// TIA Portal V20 program export: 22 tag tables, 10 data types, 20 data blocks, 41 code blocks (in call order from the OBs), 25 instance data blocks

VAR_GLOBAL   // PLC tag table "Cabinet13"
   Sz13_Column_Red AT %Q1201.2 : Bool;
   Sz13_Column_Buzzer AT %Q1201.4 : Bool;
   Sz13_Column_Green AT %Q1200.6 : Bool;
   Sz13_Column_Yellow AT %Q1201.0 : Bool;
END_VAR

VAR_GLOBAL   // PLC tag table "Cabinet14"
   Sz14_Column_Buzzer AT %Q1201.5 : Bool;
   Sz14_Column_Red AT %Q1201.3 : Bool;
   Sz14_Column_Yellow AT %Q1201.1 : Bool;
   Sz14_Column_Green AT %Q1200.7 : Bool;
END_VAR

VAR_GLOBAL   // PLC tag table "Cabinet_1"
   Sz1_St25_SenA AT %I1100.0 : Bool;
   Sz1_St25_SenB AT %I1100.1 : Bool;
   Sz1_St25_SenC AT %I1100.2 : Bool;
   Sz1_St25_SenD AT %I1100.3 : Bool;
   Sz1_St26_SenA AT %I1100.4 : Bool;
   Sz1_St26_SenB AT %I1100.5 : Bool;
   Sz1_St26_SenC AT %I1100.6 : Bool;
   Sz1_St26_SenD AT %I1100.7 : Bool;
   Sz1_St23_SenA AT %I1101.0 : Bool;
   Sz1_St23_SenB AT %I1101.1 : Bool;
   Sz1_St23_SenC AT %I1101.2 : Bool;
   Sz1_St23_SenD AT %I1101.3 : Bool;
   Sz1_St24_SenA AT %I1101.4 : Bool;
   Sz1_St24_SenB AT %I1101.5 : Bool;
   Sz1_St24_SenC AT %I1101.6 : Bool;
   Sz1_St24_SenD AT %I1101.7 : Bool;
   Sz1_Button_ST25_ST26 AT %I1102.0 : Bool;
   Sz1_Button_ST26_ST27 AT %I1102.1 : Bool;
   Sz1_Button_ST24_ST23 AT %I1102.2 : Bool;
   Sz1_Button_ST23_ST22 AT %I1102.3 : Bool;
   Sz1_Button_ST24_Seq_Backward AT %I1102.4 : Bool;
   Sz1_Button_ST24_Seq_Forward AT %I1102.5 : Bool;
   Sz1_Button_ST25_Seq_Backward AT %I1102.6 : Bool;
   Sz1_Button_ST25_Seq_Forward AT %I1102.7 : Bool;
   Sz1_Button_ST23_Seq_Forward AT %I1103.0 : Bool;
   Sz1_Button_SS_Down AT %I1103.1 : Bool;
   Sz1_Button_SS_Up AT %I1103.2 : Bool;
   Sz1_Button_SS_Drive_ST25 AT %I1103.3 : Bool;
   Sz1_Button_SS_Drive_ST24 AT %I1103.4 : Bool;
   Sz1_Button_SS_Drive_ST17 AT %I1103.5 : Bool;
   Sz1_Button_SS_Drive_ST14 AT %I1103.6 : Bool;
   "Reserved(1)" AT %I1103.7 : Bool;
   Sz1_Safety1_1 AT %I1150.0 : Bool;
   Sz13_Safety1_1 AT %I1150.1 : Bool;
   "Reserved(12)" AT %I1150.2 : Bool;
   "Reserved(13)" AT %I1150.3 : Bool;
   Sz1_Safety1_2 AT %I1150.4 : Bool;
   Sz13_Safety1_2 AT %I1150.5 : Bool;
   "Reserved(15)" AT %I1150.6 : Bool;
   "Reserved(16)" AT %I1150.7 : Bool;
   "Reserved(17)" AT %I1151.0 : Bool;
   "Reserved(18)" AT %I1151.1 : Bool;
   "Reserved(19)" AT %I1151.2 : Bool;
   "Reserved(20)" AT %I1151.3 : Bool;
   "Reserved(21)" AT %I1151.4 : Bool;
   "Reserved(22)" AT %I1151.5 : Bool;
   "Reserved(23)" AT %I1151.6 : Bool;
   "Reserved(24)" AT %I1151.7 : Bool;
   Sz1_Button_LED_ST25_ST26 AT %Q1100.0 : Bool;
   Sz1_Button_LED_ST26_ST27 AT %Q1100.1 : Bool;
   Sz1_Button_LED_ST24_ST23 AT %Q1100.2 : Bool;
   Sz1_Button_LED_ST23_ST22 AT %Q1100.3 : Bool;
   Sz1_Button_LED_Hyd_Up AT %Q1100.4 : Bool;
   Sz1_Button_LED_Hyd_Down AT %Q1100.5 : Bool;
   Sz1_Button_LED_Air_Up AT %Q1100.6 : Bool;
   Sz1_Button_LED_Air_Down AT %Q1100.7 : Bool;
   Sz1_Button_LED_Wibration AT %Q1101.0 : Bool;
   Sz1_Button_LED_SS_Down AT %Q1101.1 : Bool;
   Sz1_Button_LED_SS_Up AT %Q1101.2 : Bool;
   Sz1_Button_LED_SS_Drive_ST25 AT %Q1101.3 : Bool;
   Sz1_Button_LED_SS_Drive_ST24 AT %Q1101.4 : Bool;
   Sz1_Button_LED_SS_Drive_ST17 AT %Q1101.5 : Bool;
   Sz1_Button_LED_SS_Drive_ST14 AT %Q1101.6 : Bool;
   Reserved AT %Q1101.7 : Bool;
   Sz1_Button_LED_Centering_ST23 AT %Q1102.0 : Bool;
   Sz1_Button_LED_Centering_ST22 AT %Q1102.1 : Bool;
   "Reserved(5)" AT %Q1102.2 : Bool;
   "Reserved(6)" AT %Q1102.3 : Bool;
   Sz1_Button_LED_ST23_Seq_Backward AT %Q1102.4 : Bool;
   ST23_CNT_UPP AT %Q1102.5 : Bool;
   ST23_CNT_V1 AT %Q1102.6 : Bool;
   ST23_CNT_V2 AT %Q1102.7 : Bool;
   iSR_Distance_Value AT %IW502 : Int;
   Sz1_Button_ST23_Seq_Backward AT %I1124.0 : Bool;
   "reserved(2)" AT %I1124.1 : Bool;
   "reserved(3)" AT %I1124.2 : Bool;
   Sz1_Button_Centering_ST23 AT %I1124.3 : Bool;
   Sz1_Button_Centering_ST22 AT %I1124.4 : Bool;
   Reserved_1 AT %I1124.5 : Bool;
   Reserved_2 AT %I1124.6 : Bool;
   Reserved_3 AT %I1124.7 : Bool;
   Reserved_4 AT %I1125.0 : Bool;
   Reserved_5 AT %I1125.1 : Bool;
   Reserved_6 AT %I1125.2 : Bool;
   Reserved_7 AT %I1125.3 : Bool;
   St23_Centering_Up_2 AT %I1125.4 : Bool;
   St23_Centering_Down_2 AT %I1125.5 : Bool;
   St23_Centering_Down_1 AT %I1125.6 : Bool;
   St23_Centering_Up_1 AT %I1125.7 : Bool;
END_VAR

VAR_GLOBAL   // PLC tag table "Cabinet_10"
   Sz10_ST11_SenA AT %I2000.0 : Bool;
   Sz10_ST11_SenB AT %I2000.1 : Bool;
   Sz10_ST11_SenC AT %I2000.2 : Bool;
   Sz10_ST11_SenD AT %I2000.3 : Bool;
   Sz10_ST12_SenA AT %I2000.4 : Bool;
   Sz10_ST12_SenB AT %I2000.5 : Bool;
   Sz10_ST12_SenC AT %I2000.6 : Bool;
   Sz10_ST12_SenD AT %I2000.7 : Bool;
   Sz10_Button_ST11_ST12 AT %I2001.0 : Bool;
   Sz10_Button_ST12_ST13 AT %I2001.1 : Bool;
   "Reserved(152)" AT %I2001.2 : Bool;
   "Reserved(153)" AT %I2001.3 : Bool;
   "Reserved(154)" AT %I2001.4 : Bool;
   "Reserved(155)" AT %I2001.5 : Bool;
   "Reserved(156)" AT %I2001.6 : Bool;
   "Reserved(157)" AT %I2001.7 : Bool;
   Sz10_Safety1_1 AT %I2050.0 : Bool;
   "Reserved(158)" AT %I2050.1 : Bool;
   "Reserved(159)" AT %I2050.2 : Bool;
   "Reserved(160)" AT %I2050.3 : Bool;
   Sz10_Safety1_2 AT %I2050.4 : Bool;
   "Reserved(161)" AT %I2050.5 : Bool;
   "Reserved(162)" AT %I2050.6 : Bool;
   "Reserved(163)" AT %I2050.7 : Bool;
   "Reserved(171)" AT %I2051.0 : Bool;
   "Reserved(170)" AT %I2051.1 : Bool;
   "Reserved(169)" AT %I2051.2 : Bool;
   "Reserved(168)" AT %I2051.3 : Bool;
   "Reserved(167)" AT %I2051.4 : Bool;
   "Reserved(166)" AT %I2051.5 : Bool;
   "Reserved(165)" AT %I2051.6 : Bool;
   "Reserved(164)" AT %I2051.7 : Bool;
   Sz10_Button_LED_ST11_ST12 AT %Q2000.0 : Bool;
   Sz10_Button_LED_ST12_ST13 AT %Q2000.1 : Bool;
   "Reserved(146)" AT %Q2000.2 : Bool;
   "Reserved(147)" AT %Q2000.3 : Bool;
   "Reserved(148)" AT %Q2000.4 : Bool;
   "Reserved(149)" AT %Q2000.5 : Bool;
   "Reserved(150)" AT %Q2000.6 : Bool;
   "Reserved(151)" AT %Q2000.7 : Bool;
END_VAR

VAR_GLOBAL   // PLC tag table "Cabinet_11"
   Sz11_ST13_SenA AT %I2100.0 : Bool;
   Sz11_ST13_SenB AT %I2100.1 : Bool;
   Sz11_ST13_SenC AT %I2100.2 : Bool;
   Sz11_ST13_SenD AT %I2100.3 : Bool;
   Sz11_ST14_SenA AT %I2100.4 : Bool;
   Sz11_ST14_SenB AT %I2100.5 : Bool;
   Sz11_ST14_SenC AT %I2100.6 : Bool;
   Sz11_ST14_SenD AT %I2100.7 : Bool;
   Sz11_ST17_SenA AT %I2101.0 : Bool;
   Sz11_ST17_SenB AT %I2101.1 : Bool;
   Sz11_ST17_SenC AT %I2101.2 : Bool;
   Sz11_ST17_SenD AT %I2101.3 : Bool;
   "Reserved(188)" AT %I2101.4 : Bool;
   "Reserved(189)" AT %I2101.5 : Bool;
   "Reserved(190)" AT %I2101.6 : Bool;
   Sz11_Safety1_1 AT %I2150.0 : Bool;
   "Reserved(173)" AT %I2150.1 : Bool;
   "Reserved(174)" AT %I2150.2 : Bool;
   "Reserved(175)" AT %I2150.3 : Bool;
   Sz11_Safety1_2 AT %I2150.4 : Bool;
   "Reserved(176)" AT %I2150.5 : Bool;
   "Reserved(177)" AT %I2150.6 : Bool;
   "Reserved(178)" AT %I2150.7 : Bool;
   "Reserved(179)" AT %I2151.0 : Bool;
   "Reserved(180)" AT %I2151.1 : Bool;
   "Reserved(181)" AT %I2151.2 : Bool;
   "Reserved(182)" AT %I2151.3 : Bool;
   "Reserved(183)" AT %I2151.4 : Bool;
   "Reserved(184)" AT %I2151.5 : Bool;
   "Reserved(185)" AT %I2151.6 : Bool;
   "Reserved(186)" AT %I2151.7 : Bool;
   "Reserved(187)" AT %I2101.7 : Bool;
   Sz11_Button_ST13_ST14 AT %I2102.0 : Bool;
   Sz11_Button_SS_Down AT %I2102.1 : Bool;
   Sz11_Button_SS_Up AT %I2102.2 : Bool;
   Sz11_Button_SS_Drive_ST14 AT %I2102.3 : Bool;
   Sz11_Button_SS_Drive_ST17 AT %I2102.4 : Bool;
   Sz11_Button_SS_Drive_ST24 AT %I2102.5 : Bool;
   Sz11_Button_SS_Drive_ST25 AT %I2102.6 : Bool;
   Sz11_Button_LED_ST13_ST14 AT %Q2100.0 : Bool;
   Sz11_Button_LED_SS_Down AT %Q2100.1 : Bool;
   Sz11_Button_LED_SS_Up AT %Q2100.2 : Bool;
   Sz11_Button_LED_SS_Drive_ST14 AT %Q2100.3 : Bool;
   Sz11_Button_LED_SS_Drive_ST17 AT %Q2100.4 : Bool;
   Sz11_Button_LED_SS_Drive_ST24 AT %Q2100.5 : Bool;
   Sz11_Button_LED_SS_Drive_ST25 AT %Q2100.6 : Bool;
   "Reserved(172)" AT %Q2100.7 : Bool;
END_VAR

VAR_GLOBAL   // PLC tag table "Cabinet_2"
   Sz2_ST27_SenA AT %I1200.0 : Bool;
   Sz2_ST27_SenB AT %I1200.1 : Bool;
   Sz2_ST27_SenC AT %I1200.2 : Bool;
   Sz2_ST27_SenD AT %I1200.3 : Bool;
   Sz2_ST28_SenA AT %I1200.4 : Bool;
   Sz2_ST28_SenB AT %I1200.5 : Bool;
   Sz2_ST28_SenC AT %I1200.6 : Bool;
   Sz2_ST28_SenD AT %I1200.7 : Bool;
   Sz2_ST21_SenA AT %I1201.0 : Bool;
   Sz2_ST21_SenB AT %I1201.1 : Bool;
   Sz2_ST21_SenC AT %I1201.2 : Bool;
   Sz2_ST21_SenD AT %I1201.3 : Bool;
   Sz2_ST22_SenA AT %I1201.4 : Bool;
   Sz2_ST22_SenB AT %I1201.5 : Bool;
   Sz2_ST22_SenC AT %I1201.6 : Bool;
   Sz2_ST22_SenD AT %I1201.7 : Bool;
   Sz2_Button_ST27_ST28 AT %I1202.0 : Bool;
   Sz2_Button_ST28_ST29 AT %I1202.1 : Bool;
   Sz2_Button_ST22_ST21 AT %I1202.2 : Bool;
   Sz2_Button_ST21_ST20 AT %I1202.3 : Bool;
   Sz2_Button_Centering_ST21 AT %I1202.4 : Bool;
   Sz2_Button_Centering_ST20 AT %I1202.5 : Bool;
   "Reserved(27)" AT %I1202.6 : Bool;
   "Reserved(28)" AT %I1202.7 : Bool;
   Sz2_Safety_1_1 AT %I1250.0 : Bool;
   Sz2_Safety_1_2 AT %I1250.4 : Bool;
   "Reserved(29)" AT %I1250.1 : Bool;
   "Reserved(30)" AT %I1250.2 : Bool;
   "Reserved(31)" AT %I1250.3 : Bool;
   "Reserved(32)" AT %I1250.5 : Bool;
   "Reserved(33)" AT %I1250.6 : Bool;
   "Reserved(34)" AT %I1250.7 : Bool;
   "Reserved(35)" AT %I1251.0 : Bool;
   "Reserved(36)" AT %I1251.1 : Bool;
   "Reserved(37)" AT %I1251.2 : Bool;
   "Reserved(38)" AT %I1251.3 : Bool;
   "Reserved(39)" AT %I1251.4 : Bool;
   "Reserved(40)" AT %I1251.5 : Bool;
   "Reserved(41)" AT %I1251.6 : Bool;
   "Reserved(42)" AT %I1251.7 : Bool;
   Sz2_Button_LED_ST27_ST28 AT %Q1200.0 : Bool;
   Sz2_Button_LED_ST28_ST29 AT %Q1200.1 : Bool;
   Sz2_Button_LED_ST22_ST21 AT %Q1200.2 : Bool;
   Sz2_Button_LED_ST21_ST20 AT %Q1200.3 : Bool;
   Sz2_Button_LED_Centering_ST21 AT %Q1200.4 : Bool;
   Sz2_Button_LED_Centering_ST20 AT %Q1200.5 : Bool;
END_VAR

VAR_GLOBAL   // PLC tag table "Cabinet_3"
   Sz3_ST29_SenA AT %I1300.0 : Bool;
   Sz3_ST29_SenB AT %I1300.1 : Bool;
   Sz3_ST29_SenC AT %I1300.2 : Bool;
   Sz3_ST29_SenD AT %I1300.3 : Bool;
   Sz3_ST30_SenA AT %I1300.4 : Bool;
   Sz3_ST30_SenB AT %I1300.5 : Bool;
   Sz3_ST30_SenC AT %I1300.6 : Bool;
   Sz3_ST30_SenD AT %I1300.7 : Bool;
   Sz3_ST31_SenA AT %I1301.0 : Bool;
   Sz3_ST31_SenB AT %I1301.1 : Bool;
   Sz3_ST31_SenC AT %I1301.2 : Bool;
   Sz3_ST31_SenD AT %I1301.3 : Bool;
   Sz3_ST18_SenA AT %I1301.4 : Bool;
   Sz3_ST18_SenB AT %I1301.5 : Bool;
   Sz3_ST18_SenC AT %I1301.6 : Bool;
   Sz3_ST18_SenD AT %I1301.7 : Bool;
   Sz3_ST19_SenA AT %I1302.0 : Bool;
   Sz3_ST19_SenB AT %I1302.1 : Bool;
   Sz3_ST19_SenC AT %I1302.2 : Bool;
   Sz3_ST19_SenD AT %I1302.3 : Bool;
   Sz3_ST20_SenA AT %I1302.4 : Bool;
   Sz3_ST20_SenB AT %I1302.5 : Bool;
   Sz3_ST20_SenC AT %I1302.6 : Bool;
   Sz3_ST20_SenD AT %I1302.7 : Bool;
   Sz3_Button_ST29_ST30 AT %I1303.0 : Bool;
   Sz3_Button_ST30_ST31 AT %I1303.1 : Bool;
   Sz3_Button_ST31_ST32 AT %I1303.2 : Bool;
   Sz3_Button_ST18_ST37 AT %I1303.3 : Bool;
   Sz3_Button_ST19_ST18 AT %I1303.4 : Bool;
   Sz3_Button_ST20_ST19 AT %I1303.5 : Bool;
   Sz3_Button_Centering_ST19 AT %I1303.6 : Bool;
   Sz3_Button_Centering_ST18 AT %I1303.7 : Bool;
   Sz3_Safety1_1 AT %I1304.0 : Bool;
   Sz14_Safety1_1 AT %I1304.1 : Bool;
   "Reserved(45)" AT %I1304.2 : Bool;
   "Reserved(46)" AT %I1304.3 : Bool;
   Sz3_Safety1_2 AT %I1304.4 : Bool;
   Sz14_Safety1_2 AT %I1304.5 : Bool;
   "Reserved(48)" AT %I1304.6 : Bool;
   "Reserved(49)" AT %I1304.7 : Bool;
   "Reserved(50)" AT %I1305.0 : Bool;
   "Reserved(51)" AT %I1305.1 : Bool;
   "Reserved(52)" AT %I1305.2 : Bool;
   "Reserved(53)" AT %I1305.3 : Bool;
   "Reserved(54)" AT %I1305.4 : Bool;
   "Reserved(55)" AT %I1305.5 : Bool;
   "Reserved(56)" AT %I1305.6 : Bool;
   "Reserved(57)" AT %I1305.7 : Bool;
   Sz3_Button_LED_ST29_ST30 AT %Q1300.0 : Bool;
   Sz3_Button_LED_ST30_ST31 AT %Q1300.1 : Bool;
   Sz3_Button_LED_ST31_ST32 AT %Q1300.2 : Bool;
   Sz3_Button_LED_ST18_ST37 AT %Q1300.3 : Bool;
   Sz3_Button_LED_ST19_ST18 AT %Q1300.4 : Bool;
   Sz3_Button_LED_ST20_ST19 AT %Q1300.5 : Bool;
   Sz3_Button_LED_Centering_ST19 AT %Q1300.6 : Bool;
   Sz3_Button_LED_Centering_ST18 AT %Q1300.7 : Bool;
END_VAR

VAR_GLOBAL   // PLC tag table "Cabinet_4"
   Sz4_ST32_SenA AT %I1400.0 : Bool;
   Sz4_ST32_SenB AT %I1400.1 : Bool;
   Sz4_ST32_SenC AT %I1400.2 : Bool;
   Sz4_ST32_SenD AT %I1400.3 : Bool;
   Sz4_ST33_SenA AT %I1400.4 : Bool;
   Sz4_ST33_SenB AT %I1400.5 : Bool;
   Sz4_ST33_SenC AT %I1400.6 : Bool;
   Sz4_ST33_SenD AT %I1400.7 : Bool;
   Sz4_ST36_SenA AT %I1401.0 : Bool;
   Sz4_ST36_SenB AT %I1401.1 : Bool;
   Sz4_ST36_SenC AT %I1401.2 : Bool;
   Sz4_ST36_SenD AT %I1401.3 : Bool;
   Sz4_ST37_SenA AT %I1401.4 : Bool;
   Sz4_ST37_SenB AT %I1401.5 : Bool;
   Sz4_ST37_SenC AT %I1401.6 : Bool;
   Sz4_ST37_SenD AT %I1401.7 : Bool;
   Sz4_Button_ST32_ST33 AT %I1402.0 : Bool;
   Sz4_Button_ST33_ST34 AT %I1402.1 : Bool;
   Sz4_Button_ST36_ST38 AT %I1402.2 : Bool;
   Sz4_Button_ST37_ST36 AT %I1402.3 : Bool;
   Sz4_Button_ST34_ST33 AT %I1402.4 : Bool;
   Sz4_Button_ST38_ST36 AT %I1402.5 : Bool;
   "Reserved(60)" AT %I1402.6 : Bool;
   "Reserved(61)" AT %I1402.7 : Bool;
   Sz4_Safety1_1 AT %I1403.0 : Bool;
   Sz12_Safety1_1 AT %I1403.1 : Bool;
   "Reserved(63)" AT %I1403.2 : Bool;
   "Reserved(64)" AT %I1403.3 : Bool;
   Sz4_Safety1_2 AT %I1403.4 : Bool;
   Sz12_Safety1_2 AT %I1403.5 : Bool;
   "Reserved(66)" AT %I1403.6 : Bool;
   "Reserved(67)" AT %I1403.7 : Bool;
   "Reserved(75)" AT %I1404.0 : Bool;
   "Reserved(74)" AT %I1404.1 : Bool;
   "Reserved(73)" AT %I1404.2 : Bool;
   "Reserved(72)" AT %I1404.3 : Bool;
   "Reserved(71)" AT %I1404.4 : Bool;
   "Reserved(70)" AT %I1404.5 : Bool;
   "Reserved(69)" AT %I1404.6 : Bool;
   "Reserved(68)" AT %I1404.7 : Bool;
   Sz4_Button_LED_ST32_ST33 AT %Q1400.0 : Bool;
   Sz4_Button_LED_ST33_ST34 AT %Q1400.1 : Bool;
   Sz4_Button_LED_ST36_ST38 AT %Q1400.2 : Bool;
   Sz4_Button_LED_ST37_ST36 AT %Q1400.3 : Bool;
   Sz4_Button_LED_ST34_ST33 AT %Q1400.4 : Bool;
   Sz4_Button_LED_ST38_ST36 AT %Q1400.5 : Bool;
   "Reserved(58)" AT %Q1400.6 : Bool;
   "Reserved(59)" AT %Q1400.7 : Bool;
END_VAR

VAR_GLOBAL   // PLC tag table "Cabinet_5_6"
   Sz5_ST01_SenA AT %I1504.0 : Bool;
   Sz5_ST01_SenB AT %I1504.1 : Bool;
   Sz5_ST01_SenC AT %I1504.2 : Bool;
   Sz5_ST01_SenD AT %I1504.3 : Bool;
   Sz5_ST02_SenA AT %I1504.4 : Bool;
   Sz5_ST02_SenB AT %I1504.5 : Bool;
   Sz5_ST02_SenC AT %I1504.6 : Bool;
   Sz5_ST02_SenD AT %I1504.7 : Bool;
   Sz5_ST34_SenA AT %I1505.0 : Bool;
   Sz5_ST34_SenB AT %I1505.1 : Bool;
   Sz5_ST34_SenC AT %I1505.2 : Bool;
   Sz5_ST34_SenD AT %I1505.3 : Bool;
   Sz5_ST35_SenA AT %I1505.4 : Bool;
   Sz5_ST35_SenB AT %I1505.5 : Bool;
   Sz5_ST35_SenC AT %I1505.6 : Bool;
   Sz5_ST35_SenD AT %I1505.7 : Bool;
   Sz5_ST38_SenA AT %I1506.0 : Bool;
   Sz5_ST38_SenB AT %I1506.1 : Bool;
   Sz5_ST38_SenC AT %I1506.2 : Bool;
   Sz5_ST38_SenD AT %I1506.3 : Bool;
   Arm1_LowerClampOpen AT %I1500.0 : Bool;
   Arm1_LowerClampClosed AT %I1500.1 : Bool;
   Arm1_UpperClampOpen AT %I1500.2 : Bool;
   Arm1_UpperClampClosed AT %I1500.3 : Bool;
   Arm2_LowerClampOpen AT %I1500.4 : Bool;
   Arm2_UpperClampOpen AT %I1500.5 : Bool;
   Arm2_LowerClampClosed AT %I1500.6 : Bool;
   Arm2_UpperClampClosed AT %I1500.7 : Bool;
   S5_Arm1_BasePos AT %I1501.0 : Bool;
   S5_Arm2_BasePos AT %I1501.1 : Bool;
   S5_HydraulicStatus AT %I1501.2 : Bool;
   Arm1_Inclinometer AT %I1507.0 : "PII - JN2200";
   Arm2_Inclinometer AT %I1513.0 : "PII - JN2200";
   S6_Button_Up AT %I1501.5 : Bool;
   S5_Button_ST01_ST02 AT %I1502.0 : Bool;
   S5_Button_ST02_ST01 AT %I1502.1 : Bool;
   S5_Button_ST34_ST35 AT %I1502.2 : Bool;
   S5_Button_ST35_ST34 AT %I1502.3 : Bool;
   S5_Button_ST38_ST01 AT %I1502.4 : Bool;
   S5_Button_ST01_ST38 AT %I1502.5 : Bool;
   S5_Button_ST35 AT %I1502.6 : Bool;
   S5_Button_ST02 AT %I1502.7 : Bool;
   S5_Button_ST03 AT %I1503.0 : Bool;
   S5_Button_ST04 AT %I1503.1 : Bool;
   S5_Button_SS1_Up AT %I1503.2 : Bool;
   S5_Button_SS1_Down AT %I1503.3 : Bool;
   S5_Button_Buzz AT %I1503.4 : Bool;
   S6_Button_Buzz AT %I1503.5 : Bool;
   S5_Button_down AT %I1503.6 : Bool;
   Sz5_Estop_chA AT %I1550.0 : Bool;
   Sz6_Estop_chA AT %I1550.1 : Bool;
   Sz5_Estop_chB AT %I1550.3 : Bool;
   Sz6_Estop_chB AT %I1550.4 : Bool;
   TipHydSoftstart AT %Q2101.0 : Bool;
   TipHydContactor AT %Q2101.1 : Bool;
   UpperClampsClose AT %Q1500.0 : Bool;
   UpperClampsOpen AT %Q1500.1 : Bool;
   LowerClampsOpen AT %Q1500.2 : Bool;
   LowerClampsClose AT %Q1500.3 : Bool;
   S5_Button_LED_ST01_ST02 AT %Q1501.0 : Bool;
   S5_Button_LED_ST02_ST01 AT %Q1501.1 : Bool;
   S5_Button_LED_ST34_ST35 AT %Q1501.2 : Bool;
   S5_Button_LED_ST35_ST34 AT %Q1501.3 : Bool;
   S5_Button_LED_ST38_ST01 AT %Q1501.4 : Bool;
   S5_Button_LED_ST01_ST38 AT %Q1501.5 : Bool;
   S5_Button_LED_ST35 AT %Q1501.6 : Bool;
   S5_Button_LED_ST02 AT %Q1501.7 : Bool;
   S5_Button_LED_ST03 AT %Q1502.0 : Bool;
   S5_Button_LED_ST04 AT %Q1502.1 : Bool;
   S5_Button_LED_SS1_Up AT %Q1502.2 : Bool;
   S5_Button_LED_SS1_Down AT %Q1502.3 : Bool;
   S5_Button_LED_Buzz AT %Q1502.4 : Bool;
   S6_Button_LED_Up AT %Q1502.5 : Bool;
   S6_Button_LED_Buzz AT %Q1502.6 : Bool;
   S5_Button_LED_Down AT %Q1502.7 : Bool;
   TipArm1 AT %QW1542 : Int;
   TipArm2 AT %QW1544 : Int;
END_VAR

VAR_GLOBAL   // PLC tag table "Cabinet_7"
   Sz7_ST03_SenA AT %I1700.0 : Bool;
   Sz7_ST03_SenB AT %I1700.1 : Bool;
   Sz7_ST03_SenC AT %I1700.2 : Bool;
   Sz7_ST03_SenD AT %I1700.3 : Bool;
   Sz7_ST04_SenA AT %I1700.4 : Bool;
   Sz7_ST04_SenB AT %I1700.5 : Bool;
   Sz7_ST04_SenC AT %I1700.6 : Bool;
   Sz7_ST04_SenD AT %I1700.7 : Bool;
   Sz7_ST04_SenE AT %I1701.0 : Bool;
   Sz7_ST04_SenF AT %I1701.1 : Bool;
   Sz7_ST05_SenA AT %I1701.2 : Bool;
   Sz7_ST05_SenB AT %I1701.3 : Bool;
   Sz7_ST05_SenC AT %I1701.4 : Bool;
   Sz7_ST05_SenD AT %I1701.5 : Bool;
   "Reserved(84)" AT %I1701.6 : Bool;
   "Reserved(85)" AT %I1701.7 : Bool;
   Sz7_Button_SS_Down AT %I1702.0 : Bool;
   Sz7_Safety1_1 AT %I1750.0 : Bool;
   Sz7_Button_SS_Up AT %I1702.1 : Bool;
   Sz7_Button_SS_Drive_ST35 AT %I1702.2 : Bool;
   Sz7_Button_SS_Drive_ST02 AT %I1702.3 : Bool;
   Sz7_Button_SS_Drive_ST03 AT %I1702.4 : Bool;
   Sz7_Button_SS_Drive_ST04 AT %I1702.5 : Bool;
   Sz7_Button_ST04_ST05 AT %I1702.6 : Bool;
   Sz7_Button_ST05_ST06 AT %I1702.7 : Bool;
   "Reserved(100)" AT %I1703.0 : Bool;
   "Reserved(101)" AT %I1703.1 : Bool;
   "Reserved(102)" AT %I1703.2 : Bool;
   "Reserved(103)" AT %I1703.3 : Bool;
   "Reserved(104)" AT %I1703.4 : Bool;
   "Reserved(105)" AT %I1703.5 : Bool;
   "Reserved(106)" AT %I1703.6 : Bool;
   "Reserved(107)" AT %I1703.7 : Bool;
   "Reserved(86)" AT %I1750.1 : Bool;
   "Reserved(87)" AT %I1750.2 : Bool;
   "Reserved(88)" AT %I1750.3 : Bool;
   "Sz7-Safety1_2" AT %I1750.4 : Bool;
   "Reserved(89)" AT %I1750.5 : Bool;
   "Reserved(90)" AT %I1750.6 : Bool;
   "Reserved(91)" AT %I1750.7 : Bool;
   "Reserved(92)" AT %I1751.0 : Bool;
   "Reserved(93)" AT %I1751.1 : Bool;
   "Reserved(94)" AT %I1751.2 : Bool;
   "Reserved(95)" AT %I1751.3 : Bool;
   "Reserved(96)" AT %I1751.4 : Bool;
   "Reserved(97)" AT %I1751.5 : Bool;
   "Reserved(98)" AT %I1751.6 : Bool;
   "Reserved(99)" AT %I1751.7 : Bool;
   Sz7_Button_LED_SS_Down AT %Q1700.0 : Bool;
   Sz7_Button_LED_SS_Up AT %Q1700.1 : Bool;
   Sz7_Button_LED_SS_Drive_ST35 AT %Q1700.2 : Bool;
   Sz7_Button_LED_SS_Drive_ST02 AT %Q1700.3 : Bool;
   Sz7_Button_LED_SS_Drive_ST03 AT %Q1700.4 : Bool;
   Sz7_Button_LED_SS_Drive_ST04 AT %Q1700.5 : Bool;
   Sz7_Button_LED_ST04_ST05 AT %Q1700.6 : Bool;
   Sz7_Button_LED_ST05_ST06 AT %Q1700.7 : Bool;
   "Reserved(76)" AT %Q1701.0 : Bool;
   "Reserved(77)" AT %Q1701.1 : Bool;
   "Reserved(78)" AT %Q1701.2 : Bool;
   "Reserved(79)" AT %Q1701.3 : Bool;
   "Reserved(80)" AT %Q1701.4 : Bool;
   "Reserved(81)" AT %Q1701.5 : Bool;
   "Reserved(82)" AT %Q1701.6 : Bool;
   "Reserved(83)" AT %Q1701.7 : Bool;
END_VAR

VAR_GLOBAL   // PLC tag table "Cabinet_8"
   Sz8_ST06_SenA AT %I1800.0 : Bool;
   Sz8_ST06_SenB AT %I1800.1 : Bool;
   Sz8_ST06_SenC AT %I1800.2 : Bool;
   Sz8_ST06_SenD AT %I1800.3 : Bool;
   Sz8_ST07_SenA AT %I1800.4 : Bool;
   Sz8_ST07_SenB AT %I1800.5 : Bool;
   Sz8_ST07_SenC AT %I1800.6 : Bool;
   Sz8_ST07_SenD AT %I1800.7 : Bool;
   Sz8_ST08_SenA AT %I1801.0 : Bool;
   Sz8_ST08_SenB AT %I1801.1 : Bool;
   Sz8_ST08_SenC AT %I1801.2 : Bool;
   Sz8_ST08_SenD AT %I1801.3 : Bool;
   Sz8_Button_ST06_ST07 AT %I1801.4 : Bool;
   Sz8_Button_ST07_ST08 AT %I1801.5 : Bool;
   Sz8_Button_ST08_ST09 AT %I1801.6 : Bool;
   Sz8_Button_Centering_ST08 AT %I1801.7 : Bool;
   Sz8_Safety1_1 AT %I1850.0 : Bool;
   "Reserved(112)" AT %I1850.1 : Bool;
   "Reserved(113)" AT %I1850.2 : Bool;
   "Reserved(114)" AT %I1850.3 : Bool;
   Sz8_Safety1_2 AT %I1850.4 : Bool;
   "Reserved(115)" AT %I1850.5 : Bool;
   "Reserved(116)" AT %I1850.6 : Bool;
   "Reserved(117)" AT %I1850.7 : Bool;
   "Reserved(118)" AT %I1851.0 : Bool;
   "Reserved(119)" AT %I1851.1 : Bool;
   "Reserved(120)" AT %I1851.2 : Bool;
   "Reserved(121)" AT %I1851.3 : Bool;
   "Reserved(122)" AT %I1851.4 : Bool;
   "Reserved(123)" AT %I1851.5 : Bool;
   "Reserved(124)" AT %I1851.6 : Bool;
   "Reserved(125)" AT %I1851.7 : Bool;
   Sz8_Button_LED_ST06_ST07 AT %Q1800.0 : Bool;
   Sz8_Button_LED_ST07_ST08 AT %Q1800.1 : Bool;
   Sz8_Button_LED_ST08_ST09 AT %Q1800.2 : Bool;
   Sz8_Button_LED_Centering_ST08 AT %Q1800.3 : Bool;
   Sz8_Column_Green AT %Q1800.4 : Bool;
   Sz8_Column_Yellow AT %Q1800.5 : Bool;
   Sz8_Column_Red AT %Q1800.6 : Bool;
   Sz8_Column_Buzzer AT %Q1800.7 : Bool;
END_VAR

VAR_GLOBAL   // PLC tag table "Cabinet_9"
   Sz9_ST09_SenA AT %I1900.0 : Bool;
   Sz9_ST09_SenB AT %I1900.1 : Bool;
   Sz9_ST09_SenC AT %I1900.2 : Bool;
   Sz9_ST09_SenD AT %I1900.3 : Bool;
   Sz9_ST10_SenA AT %I1900.4 : Bool;
   Sz9_ST10_SenB AT %I1900.5 : Bool;
   Sz9_ST10_SenC AT %I1900.6 : Bool;
   Sz9_ST10_SenD AT %I1900.7 : Bool;
   Sz9_Button_ST09_ST10 AT %I1901.0 : Bool;
   Sz9_Button_ST10_ST11 AT %I1901.1 : Bool;
   Sz9_Oil_Error AT %I1901.2 : Bool;
   Sz9_Oil_Pump_Status AT %I1901.3 : Bool;
   "Reserved(128)" AT %I1901.4 : Bool;
   "Reserved(129)" AT %I1901.5 : Bool;
   "Reserved(130)" AT %I1901.6 : Bool;
   "Reserved(131)" AT %I1901.7 : Bool;
   Sz9_Safety1_1 AT %I1950.0 : Bool;
   Sz9_Safety1_2 AT %I1950.4 : Bool;
   "Reserved(132)" AT %I1950.1 : Bool;
   "Reserved(133)" AT %I1950.2 : Bool;
   "Reserved(134)" AT %I1950.3 : Bool;
   "Reserved(135)" AT %I1950.5 : Bool;
   "Reserved(136)" AT %I1950.6 : Bool;
   "Reserved(137)" AT %I1950.7 : Bool;
   "Reserved(138)" AT %I1951.0 : Bool;
   "Reserved(139)" AT %I1951.1 : Bool;
   "Reserved(140)" AT %I1951.2 : Bool;
   "Reserved(141)" AT %I1951.3 : Bool;
   "Reserved(142)" AT %I1951.4 : Bool;
   "Reserved(143)" AT %I1951.5 : Bool;
   "Reserved(144)" AT %I1951.6 : Bool;
   "Reserved(145)" AT %I1951.7 : Bool;
   Sz9_Button_LED_ST09_ST10 AT %Q1900.0 : Bool;
   Sz9_Button_LED_ST10_ST11 AT %Q1900.1 : Bool;
   Sz9_Oil_Main_Valve AT %Q1900.2 : Bool;
   Sz9_Oil_Preparation_Valve AT %Q1900.3 : Bool;
   Sz9_Oil_Open_Nozzle AT %Q1900.4 : Bool;
   Sz9_Oil_Pump AT %Q1900.5 : Bool;
   Sz9_Oil_Pump_Volume AT %QW1901 : Int;
END_VAR

VAR_GLOBAL   // PLC tag table "CentralShifter"
   iCS_SensorHoming_Left AT %I3000.0 : Bool;
   iCS_SensorHoming_Right AT %I3000.2 : Bool;
   CS_R1_Sen_Drv_1 AT %I3100.0 : Bool;
   CS_R1_Sen_Drv_2 AT %I3100.1 : Bool;
   CS_R1_Sen_Drv_3 AT %I3100.2 : Bool;
   CS_R1_Sen_Drv_4 AT %I3100.3 : Bool;
   CS_R1_Sen_Val1_Up AT %I3100.4 : Bool;
   CS_R1_Sen_Val1_Down AT %I3100.5 : Bool;
   CS_R1_Sen_Val2_Up AT %I3100.6 : Bool;
   CS_R1_Sen_Val2_Down AT %I3100.7 : Bool;
   CS_R1_Hyd_Filtr AT %I3101.0 : Bool;
   CS_R1_Hyd_Empty AT %I3101.1 : Bool;
   CS_R1_Safety1_1 AT %I3150.0 : Bool;
   CS_R1_Safety2_1 AT %I3150.1 : Bool;
   CS_R1_Safety3_1 AT %I3150.2 : Bool;
   CS_R1_Safety4_1 AT %I3150.3 : Bool;
   CS_R1_Safety1_2 AT %I3150.4 : Bool;
   CS_R1_Safety2_2 AT %I3150.5 : Bool;
   CS_R1_Safety3_2 AT %I3150.6 : Bool;
   CS_R1_Safety4_2 AT %I3150.7 : Bool;
   CS_R1_Valve_Up AT %Q3100.0 : Bool;
   CS_R1_Valve_Down AT %Q3100.1 : Bool;
   CS_R1_Hydraulic_Unit AT %Q3100.2 : Bool;
   iCS_L_Distance_Value AT %IW3102 : Int;
   CS_R2_Sen_Drv_1 AT %I3200.0 : Bool;
   CS_R2_Sen_Drv_2 AT %I3200.1 : Bool;
   CS_R2_Sen_Drv_3 AT %I3200.2 : Bool;
   CS_R2_Sen_Drv_4 AT %I3200.3 : Bool;
   CS_R2_Sen_Val1_Up AT %I3200.4 : Bool;
   CS_R2_Sen_Val1_Down AT %I3200.5 : Bool;
   CS_R2_Sen_Val2_Up AT %I3200.6 : Bool;
   CS_R2_Sen_Val2_Down AT %I3200.7 : Bool;
   CS_R2_Hyd_Filtr AT %I3201.0 : Bool;
   CS_R2_Hyd_Empty AT %I3201.1 : Bool;
   iCS_R_Distance_Value AT %IW3202 : Int;
   CS_R2_Safety1_1 AT %I3250.0 : Bool;
   CS_R2_Safety2_1 AT %I3250.1 : Bool;
   CS_R2_Safety3_1 AT %I3250.2 : Bool;
   CS_R2_Safety4_1 AT %I3250.3 : Bool;
   CS_R2_Safety1_2 AT %I3250.4 : Bool;
   CS_R2_Safety2_2 AT %I3250.5 : Bool;
   CS_R2_Safety3_2 AT %I3250.6 : Bool;
   CS_R2_Safety4_2 AT %I3250.7 : Bool;
   CS_R2_Valve_Up AT %Q3200.0 : Bool;
   CS_R2_Valve_Down AT %Q3200.1 : Bool;
   CS_R2_Hydraulic_Unit AT %Q3200.2 : Bool;
END_VAR

VAR_GLOBAL   // PLC tag table "Default tag table"
   SAFETY_TEST AT %M200.0 : Bool;
   Tag_1 AT %M200.1 : Bool;
   Tag_3 AT %M2000.0 : Bool;
   Tag_4 AT %M2000.1 : Bool;
   armsMainValve AT %Q1557.0 : Bool;
   clampsMainValve AT %Q1557.1 : Bool;
   Tag_5 AT %M2001.0 : Bool;
   Tag_6 AT %M2001.1 : Bool;
   Tag_7 AT %M2001.3 : Bool;
   Tag_8 AT %M2001.2 : Bool;
   Tag_9 AT %M222.2 : Bool;
   SS2_R1_STO AT %Q150.0 : Bool;
   Tag_11 AT %M222.3 : Bool;
   Tag_10 AT %M212.0 : Bool;
   Tag_12 AT %M500.0 : Bool;
   Tag_13 AT %M500.1 : Bool;
   Tag_14 AT %M500.2 : Bool;
   Tag_15 AT %M501.0 : Bool;
   Tag_16 AT %M501.1 : Bool;
   TipHydContactorFB AT %I2105.0 : Bool;
   S2_R2_STO AT %Q169.0 : Bool;
   Tag_17 AT %M3000.0 : Bool;
   Tag_18 AT %M3000.1 : Bool;
   Tag_2 AT %M222.4 : Bool;
   Tag_19 AT %M222.5 : Bool;
   CS_Drive_PL_Actor_Interface_AddressIn AT %I50.0 : "PD_TEL105_IN";
   CS_Drive_PP_Actor_Interface_AddressIn AT %I18.0 : "PD_TEL105_IN";
   CS_Drive_TL_Actor_Interface_AddressIn AT %I102.0 : "PD_TEL105_IN";
   CS_Drive_TP_Actor_Interface_AddressIn AT %I76.0 : "PD_TEL105_IN";
   "CS_Drive_PL_Actor_Interface_AddressIn(1)" AT %I50.0 : "PD_TEL1_IN";
   CS_Drive_PL_Actor_Interface_AddressOut AT %Q50.0 : "PD_TEL105_OUT";
   CS_Drive_PP_Actor_Interface_AddressOut AT %Q18.0 : "PD_TEL105_OUT";
   CS_Drive_TL_Actor_Interface_AddressOut AT %Q102.0 : "PD_TEL105_OUT";
   CS_Drive_TP_Actor_Interface_AddressOut AT %Q76.0 : "PD_TEL105_OUT";
   "CS_Drive_PL_Actor_Interface_AddressOut(1)" AT %Q50.0 : "PD_TEL1_OUT";
   Clock_Byte AT %MB1000 : Byte;
   Clock_10Hz AT %M1000.0 : Bool;
   Clock_5Hz AT %M1000.1 : Bool;
   "Clock_2.5Hz" AT %M1000.2 : Bool;
   Clock_2Hz AT %M1000.3 : Bool;
   "Clock_1.25Hz" AT %M1000.4 : Bool;
   Clock_1Hz AT %M1000.5 : Bool;
   "Clock_0.625Hz" AT %M1000.6 : Bool;
   "Clock_0.5Hz" AT %M1000.7 : Bool;
   Tag_20 AT %M600.0 : Bool;
   Tag_22 AT %Q600.3 : Bool;
   SS1_R1_STO AT %Q122.0 : Bool;
   SS1_R1_ACK_STO AT %Q122.7 : Bool;
   SS1_R2_STO AT %Q131.0 : Bool;
   SS1_R2_ACK_STO AT %Q131.7 : Bool;
   Tag_23 AT %Q400.3 : Bool;
   Tag_24 AT %M666.0 : Bool;
   "SS1_R1_STO(1)" AT %Q896.0 : Bool;
   "SS1_R2_STO(1)" AT %Q915.0 : Bool;
   Tag_21 AT %M2222.0 : Bool;
   SpeedAxis_1_Actor_Interface_AddressIn AT %I345.0 : "PD_TEL1_IN";
   SpeedAxis_1_Actor_Interface_AddressOut AT %Q344.0 : "PD_TEL1_OUT";
   Tag_25 AT %M999.0 : Bool;
   Tag_26 AT %M999.1 : Bool;
   Tag_27 AT %M999.2 : Bool;
   "CS_Drive_PL_Actor_Interface_AddressIn(3)" AT %I120.0 : "PD_TEL105_IN";
   "CS_Drive_PL_Actor_Interface_AddressOut(3)" AT %Q120.0 : "PD_TEL105_OUT";
   "CS_Drive_PL_Actor_Interface_AddressIn(4)" AT %I1157.0 : "PD_TEL3_IN";
   "CS_Drive_PL_Actor_Interface_AddressOut(4)" AT %Q1157.0 : "PD_TEL3_OUT";
   Tag_28 AT %Q1175.0 : Bool;
   Tag_29 AT %Q1175.1 : Bool;
   Tag_30 AT %M444.0 : Bool;
   "CS_Drive_PP_Actor_Interface_AddressIn(1)" AT %I120.0 : "PD_TEL3_IN";
   "CS_Drive_PP_Actor_Interface_AddressOut(1)" AT %Q0.0 : "PD_TEL3_OUT";
   STO_CS_PL AT %Q393.0 : Bool;
   "CS_Drive_PL_Actor_Interface_AddressIn(5)" AT %I1177.0 : "PD_TEL105_IN";
   "CS_Drive_PL_Actor_Interface_AddressOut(5)" AT %Q1177.0 : "PD_TEL105_OUT";
   "CS_Drive_PP_Actor_Interface_AddressIn(2)" AT %I1157.0 : "PD_TEL105_IN";
   "CS_Drive_PP_Actor_Interface_AddressOut(2)" AT %Q1157.0 : "PD_TEL105_OUT";
   "CS_Drive_TL_Actor_Interface_AddressIn(1)" AT %I1203.0 : "PD_TEL105_IN";
   "CS_Drive_TL_Actor_Interface_AddressOut(1)" AT %Q1203.0 : "PD_TEL105_OUT";
   "CS_Drive_TP_Actor_Interface_AddressIn(1)" AT %I1223.0 : "PD_TEL105_IN";
   "CS_Drive_TP_Actor_Interface_AddressOut(1)" AT %Q1223.0 : "PD_TEL105_OUT";
   STO_CS_PP AT %Q643.0 : Bool;
   STO_CS_TP AT %Q1140.0 : Bool;
   STO_CS_TL AT %Q1243.0 : Bool;
   Tag_33 AT %M777.0 : Bool;
   Tag_34 AT %M777.1 : Bool;
   Tag_35 AT %M777.3 : Bool;
   Tag_36 AT %M777.5 : Bool;
   Tag_37 AT %M777.6 : Bool;
   Tag_38 AT %M777.7 : Bool;
   Tag_39 AT %M778.1 : Bool;
   Tag_40 AT %M888.0 : Bool;
   Tag_41 AT %M779.0 : Bool;
   CS_QR_Reader AT %IW5002 : Word;
   QR_Reader AT %ID5000 : DWord;
   Tag_43 AT %M832.0 : Bool;
   STO_CS_R1 AT %Q226.0 : Bool;
   STO_CS_R2 AT %Q245.0 : Bool;
   Tag_31 AT %IW5000 : Word;
   STO_CSM1 AT %Q188.0 : Bool;
   STO_CSM2 AT %Q207.0 : Bool;
   Tag_32 AT %M657.4 : Bool;
   CC_Vibrating_Unit_1_Actor_Interface_AddressIn AT %I446.0 : "PD_TEL1_IN";
   CC_Vibrating_Unit_1_Actor_Interface_AddressOut AT %Q445.0 : "PD_TEL1_OUT";
   CC_Vibrating_Unit_3_Actor_Interface_AddressIn AT %I544.0 : "PD_TEL1_IN";
   CC_Vibrating_Unit_3_Actor_Interface_AddressOut AT %Q544.0 : "PD_TEL1_OUT";
   CC_Vibrating_Unit_2_Actor_Interface_AddressIn AT %I495.0 : "PD_TEL1_IN";
   CC_Vibrating_Unit_2_Actor_Interface_AddressOut AT %Q494.0 : "PD_TEL1_OUT";
   Tag_42 AT %M946.0 : Bool;
   Tag_44 AT %MB856 : Byte;
   STO_MST30B AT %Q1115.0 : Bool;
   STO_MST29 AT %Q1257.0 : Bool;
   Tag_45 AT %M442.0 : Bool;
   Tag_46 AT %M445.0 : Bool;
   Tag_47 AT %M558.4 : Bool;
   Tag_48 AT %M487.4 : Bool;
   Tag_49 AT %M699.1 : Bool;
   Tag_50 AT %M467.0 : Bool;
   Tag_51 AT %M788.5 : Bool;
   Tag_52 AT %M376.4 : Bool;
   Tag_53 AT %M35.4 : Bool;
   Tag_54 AT %M323.3 : Bool;
   Tag_55 AT %M452.3 : Bool;
   Tag_56 AT %M669.3 : Bool;
   Tag_57 AT %M100.3 : Bool;
   Tag_58 AT %Q2250.1 : Bool;
   Tag_59 AT %M836.4 : Bool;
   Tag_60 AT %M816.0 : Bool;
   Tag_61 AT %M997.0 : Bool;
   Tag_62 AT %M100.0 : Bool;
   Tag_63 AT %M899.6 : Bool;
   CS_Drive_PL_Actor_Interface_TorqueDataAddressIn AT %I1294.0 : "PD_TEL750_IN";
   CS_Drive_PL_Actor_Interface_TorqueDataAddressOut AT %Q1294.0 : "PD_TEL750_OUT";
   CS_Drive_PP_Actor_Interface_TorqueDataAddressIn AT %I1420.0 : "PD_TEL750_IN";
   CS_Drive_PP_Actor_Interface_TorqueDataAddressOut AT %Q1420.0 : "PD_TEL750_OUT";
   CS_Drive_TL_Actor_Interface_TorqueDataAddressIn AT %I1426.0 : "PD_TEL750_IN";
   CS_Drive_TL_Actor_Interface_TorqueDataAddressOut AT %Q1426.0 : "PD_TEL750_OUT";
   CS_Drive_TP_Actor_Interface_TorqueDataAddressIn AT %I1432.0 : "PD_TEL750_IN";
   CS_Drive_TP_Actor_Interface_TorqueDataAddressOut AT %Q1432.0 : "PD_TEL750_OUT";
   Tag_64 AT %M655.3 : Bool;
   Tag_65 AT %M599.1 : Bool;
   Tag_66 AT %M476.2 : Bool;
   Tag_67 AT %M888.2 : Bool;
   Tag_68 AT %M444.3 : Bool;
   Tag_69 AT %M398.4 : Bool;
   Tag_70 AT %M1333.0 : Bool;
   Tag_71 AT %M611.2 : Bool;
   Tag_72 AT %M611.3 : Bool;
   Tag_73 AT %M833.4 : Bool;
   Tag_74 AT %M881.1 : Bool;
   Tag_75 AT %M71.0 : Bool;
   Tag_76 AT %M727.1 : Bool;
END_VAR

VAR_GLOBAL   // PLC tag table "Motors"
   STO_MST1 AT %Q357.0 : Bool;
   STO_MST38 AT %Q366.0 : Bool;
   STO_MST35 AT %Q264.0 : Bool;
   STO_MST34 AT %Q273.0 : Bool;
   STO_MST33a AT %Q282.0 : Bool;
   STO_MST33b AT %Q291.0 : Bool;
   STO_MST32 AT %Q327.0 : Bool;
   STO_MST31 AT %Q318.0 : Bool;
   STO_MST30a AT %Q336.0 : Bool;
   STO_MST36a AT %Q375.0 : Bool;
   STO_MST36b AT %Q384.0 : Bool;
   STO_MST37 AT %Q418.0 : Bool;
   STO_MST18 AT %Q437.0 : Bool;
   STO_MST19a AT %Q467.0 : Bool;
   STO_MST4a AT %Q486.0 : Bool;
   STO_MST4b AT %Q557.0 : Bool;
   STO_MST5 AT %Q576.0 : Bool;
   STO_MST6a AT %Q634.0 : Bool;
   STO_MST6b AT %Q667.0 : Bool;
   STO_MST7 AT %Q686.0 : Bool;
   STO_MST8 AT %Q705.0 : Bool;
   STO_MST9a AT %Q724.0 : Bool;
   STO_MST9b AT %Q743.0 : Bool;
   STO_MST10 AT %Q762.0 : Bool;
   STO_MST11 AT %Q781.0 : Bool;
   STO_MST12a AT %Q801.0 : Bool;
   STO_MST12b AT %Q820.0 : Bool;
   STO_MST13 AT %Q839.0 : Bool;
   STO_MST14 AT %Q858.0 : Bool;
   STO_MST17 AT %Q877.0 : Bool;
   STO_Mst19b AT %Q934.0 : Bool;
   STO_Mst20 AT %Q953.0 : Bool;
   STO_Mst21 AT %Q991.0 : Bool;
   STO_Mst22a AT %Q972.0 : Bool;
   STO_Mst22b AT %Q1010.0 : Bool;
   STO_Mst23a AT %Q1067.0 : Bool;
   STO_Mst23b AT %Q1029.0 : Bool;
   STO_Mst24a AT %Q1048.0 : Bool;
   STO_Mst24b AT %Q1086.0 : Bool;
   STO_MST1a AT %Q1131.0 : Bool;
   STO_Mst25a AT %Q1311.0 : Bool;
   STO_Mst25b AT %Q1330.0 : Bool;
   STO_Mst26 AT %Q1349.0 : Bool;
   STO_Mst27a AT %Q1368.0 : Bool;
   STO_Mst27b AT %Q1387.0 : Bool;
   STO_MST28 AT %Q1275.0 : Bool;
END_VAR

VAR_GLOBAL   // PLC tag table "SS0"
   SS0_Column_Green AT %Q2101.4 : Bool;
   SS0_Column_Yellow AT %Q2101.5 : Bool;
   SS0_Column_Red AT %Q2101.6 : Bool;
   SS0_Column_Buzzer AT %Q2101.7 : Bool;
END_VAR

VAR_GLOBAL   // PLC tag table "SS2"
   SS2_Column_Buzzer AT %Q2203.7 : Bool;
   SS2_Column_Red AT %Q2203.6 : Bool;
   SS2_Column_Yellow AT %Q2203.5 : Bool;
   SS2_Column_Green AT %Q2203.4 : Bool;
   ST23_Hydraulic_Rollers_Down AT %Q2200.0 : Bool;
   ST23_Hydraulic_Rollers_Up AT %Q2200.1 : Bool;
   ST23_Modules_Up AT %Q2200.2 : Bool;
   reserve AT %Q2200.3 : Bool;
   "reserve(1)" AT %Q2200.4 : Bool;
   ST24_Hydraulic_Rollers_Down AT %Q2200.5 : Bool;
   ST24_Hydraulic_Rollers_Up AT %Q2200.6 : Bool;
   ST24_Modules_Up AT %Q2200.7 : Bool;
   "reserve(2)" AT %Q2201.0 : Bool;
   "reserve(3)" AT %Q2201.1 : Bool;
   ST25_Hydraulic_Rollers_Down AT %Q2201.2 : Bool;
   ST25_Hydraulic_Rollers_Up AT %Q2201.3 : Bool;
   ST25_Modules_Up AT %Q2201.4 : Bool;
   "reserve(4)" AT %Q2201.5 : Bool;
   "reserve(5)" AT %Q2201.6 : Bool;
   ST23_MOD1_Sen11 AT %I2200.0 : Bool;
   ST23_MOD1_Sen12 AT %I2200.1 : Bool;
   ST23_MOD1_Sen21 AT %I2200.2 : Bool;
   ST23_MOD1_Sen22 AT %I2200.3 : Bool;
   ST23_MOD2_Sen11 AT %I2200.4 : Bool;
   ST23_MOD2_Sen12 AT %I2200.5 : Bool;
   ST23_MOD2_Sen21 AT %I2200.6 : Bool;
   ST23_MOD2_Sen22 AT %I2200.7 : Bool;
   ST23_MOD3_Sen11 AT %I2201.0 : Bool;
   ST23_MOD3_Sen12 AT %I2201.1 : Bool;
   ST23_MOD3_Sen21 AT %I2201.2 : Bool;
   ST23_MOD3_Sen22 AT %I2201.3 : Bool;
   ST23_PAL_Sen11 AT %I2201.4 : Bool;
   ST23_PAL_Sen12 AT %I2201.5 : Bool;
   ST23_PAL_Sen21 AT %I2201.6 : Bool;
   ST23_PAL_Sen22 AT %I2201.7 : Bool;
   ST24_MOD1_Sen11 AT %I2202.0 : Bool;
   ST24_MOD1_Sen12 AT %I2202.1 : Bool;
   ST24_MOD1_Sen21 AT %I2202.2 : Bool;
   ST24_MOD1_Sen22 AT %I2202.3 : Bool;
   ST24_MOD2_Sen11 AT %I2202.4 : Bool;
   ST24_MOD2_Sen12 AT %I2202.5 : Bool;
   ST24_MOD2_Sen21 AT %I2202.6 : Bool;
   ST24_MOD2_Sen22 AT %I2202.7 : Bool;
   ST24_MOD3_Sen11 AT %I2203.0 : Bool;
   ST24_MOD3_Sen12 AT %I2203.1 : Bool;
   ST24_MOD3_Sen21 AT %I2203.2 : Bool;
   ST24_MOD3_Sen22 AT %I2203.3 : Bool;
   ST24_PAL_Sen11 AT %I2203.4 : Bool;
   ST24_PAL_Sen12 AT %I2203.5 : Bool;
   ST24_PAL_Sen21 AT %I2203.6 : Bool;
   ST24_PAL_Sen22 AT %I2203.7 : Bool;
   ST23_Drivers_Rollers_Up AT %Q2202.0 : Bool;
   ST24_Drivers_Rollers_Up AT %Q2202.1 : Bool;
   ST25_Drivers_Rollers_Up AT %Q2202.2 : Bool;
   ST25_MOD1_Sen11 AT %I2204.0 : Bool;
   ST25_MOD1_Sen12 AT %I2204.1 : Bool;
   ST25_MOD1_Sen21 AT %I2204.2 : Bool;
   ST25_MOD1_Sen22 AT %I2204.3 : Bool;
   ST25_MOD2_Sen11 AT %I2204.4 : Bool;
   ST25_MOD2_Sen12 AT %I2204.5 : Bool;
   ST25_MOD2_Sen21 AT %I2204.6 : Bool;
   ST25_MOD2_Sen22 AT %I2204.7 : Bool;
   ST25_MOD3_Sen11 AT %I2205.0 : Bool;
   ST25_MOD3_Sen12 AT %I2205.1 : Bool;
   ST25_MOD3_Sen21 AT %I2205.2 : Bool;
   ST25_MOD3_Sen22 AT %I2205.3 : Bool;
   ST25_PAL_Sen11 AT %I2205.4 : Bool;
   ST25_PAL_Sen12 AT %I2205.5 : Bool;
   ST25_PAL_Sen21 AT %I2205.6 : Bool;
   ST25_PAL_Sen22 AT %I2205.7 : Bool;
   ST23_25_Y0 AT %Q2250.0 : Bool;
   Estop_SS2_ChA AT %I2255.0 : Bool;
   Estop_SS2_ChB AT %I2255.4 : Bool;
   ST23_DR_a_Up AT %I2206.0 : Bool;
   ST23_DR_a_Down AT %I2206.1 : Bool;
   ST23_DR_b_Up AT %I2206.2 : Bool;
   ST23_DR_b_Down AT %I2206.3 : Bool;
   ST24_DR_a_Up AT %I2206.4 : Bool;
   ST24_DR_a_Down AT %I2206.5 : Bool;
   ST24_DR_b_Up AT %I2206.6 : Bool;
   ST24_DR_b_Down AT %I2206.7 : Bool;
   ST25_DR_a_Up AT %I2207.0 : Bool;
   ST25_DR_a_Down AT %I2207.1 : Bool;
   ST25_DR_b_Up AT %I2207.2 : Bool;
   ST25_DR_b_Down AT %I2207.3 : Bool;
   ST23_MOD1_Wib_Contactor AT %Q2202.3 : Bool;
   ST25_MOD1_Wib_Contactor AT %Q2202.4 : Bool;
   ST24_MOD1_Wib_Contactor AT %Q2202.5 : Bool;
   ST23_MOD2_Wib_Contactor AT %Q2202.6 : Bool;
   ST25_MOD2_Wib_Contactor AT %Q2202.7 : Bool;
   ST24_MOD2_Wib_Contactor AT %Q2203.0 : Bool;
   ST23_MOD3_Wib_Contactor AT %Q2203.1 : Bool;
   ST25_MOD3_Wib_Contactor AT %Q2203.2 : Bool;
   ST24_MOD3_Wib_Contactor AT %Q2203.3 : Bool;
END_VAR

VAR_GLOBAL   // PLC tag table "LSql_UserConstants"
END_VAR
VAR_GLOBAL CONSTANT   // user constants
   LSQL_NUMBER_OF_COLUMNS_MAX : UInt := 9;   // upper bound of array for expected columns (zero-based!)
   LSQL_NUMBER_OF_ROWS_MAX : UInt := 9;   // upper bound of array for expected rows (zero-based!)
   LSQL_NUMBER_OF_ROWS_PER_CYCLE : USInt := 0;   // number of rows to be deserialized per cycle (0 = all at once)
END_VAR

VAR_GLOBAL   // PLC tag table "S1_R1"
   S1_R1_Sen_Drv_1 AT %I300.0 : Bool;
   S1_R1_Sen_Drv_2 AT %I300.1 : Bool;
   S1_R1_Sen_Drv_3 AT %I300.2 : Bool;
   S1_R1_Sen_Drv_4 AT %I300.3 : Bool;
   S1_R1_Sen_Val1_Up AT %I300.4 : Bool;
   S1_R1_Sen_Val1_Down AT %I300.5 : Bool;
   S1_R1_Sen_Val2_Up AT %I300.6 : Bool;
   S1_R1_Sen_Val2_Down AT %I300.7 : Bool;
   S1_R1_Hyd_Filtr AT %I301.0 : Bool;
   S1_R1_Hyd_Empty AT %I301.1 : Bool;
   S1_R1_Safety1_1 AT %I350.0 : Bool;
   S1_R1_Safety2_1 AT %I350.1 : Bool;
   S1_R1_Safety3_1 AT %I350.2 : Bool;
   S1_R1_Safety4_1 AT %I350.3 : Bool;
   S1_R1_Safety1_2 AT %I351.0 : Bool;
   S1_R1_Safety2_2 AT %I351.1 : Bool;
   S1_R1_Safety3_2 AT %I351.2 : Bool;
   S1_R1_Safety4_2 AT %I351.3 : Bool;
   S1_R1_Valve_Up AT %Q300.0 : Bool;
   S1_R1_Valve_Down AT %Q300.1 : Bool;
   S1_R1_Hydraulic_Unit AT %Q300.2 : Bool;
   iS1L_Distance_Value AT %IW302 : Int;
END_VAR

VAR_GLOBAL   // PLC tag table "S1_R2"
   S1_R2_Safety1_1 AT %I450.0 : Bool;
   S1_R2_Safety2_1 AT %I450.1 : Bool;
   S1_R2_Safety3_1 AT %I450.2 : Bool;
   S1_R2_Safety4_1 AT %I450.3 : Bool;
   S1_R2_Safety1_2 AT %I451.0 : Bool;
   S1_R2_Safety2_2 AT %I451.1 : Bool;
   S1_R2_Safety3_2 AT %I451.2 : Bool;
   S1_R2_Safety4_2 AT %I451.3 : Bool;
   S1_R2_Valve_Up AT %Q400.0 : Bool;
   S1_R2_Valve_Down AT %Q400.1 : Bool;
   S1_R2_Sen_Drv_1 AT %I400.0 : Bool;
   S1_R2_Sen_Drv_2 AT %I400.1 : Bool;
   S1_R2_Sen_Drv_3 AT %I400.2 : Bool;
   S1_R2_Sen_Drv_4 AT %I400.3 : Bool;
   S1_R2_Sen_Val1_Up AT %I400.4 : Bool;
   S1_R2_Sen_Val1_Down AT %I400.5 : Bool;
   S1_R2_Sen_Val2_Up AT %I400.6 : Bool;
   S1_R2_Sen_Val2_Down AT %I400.7 : Bool;
   S1_R2_Hyd_Filtr AT %I401.0 : Bool;
   S1_R2_Hyd_Empty AT %I401.1 : Bool;
   S1_R2_Hydraulic_Unit AT %Q400.2 : Bool;
   iS1R_Distance_Value AT %IW402 : Int;
END_VAR

VAR_GLOBAL   // PLC tag table "S2_R1"
   S2_R1_Safety1_1 AT %I550.0 : Bool;
   S2_R1_Safety2_1 AT %I550.1 : Bool;
   S2_R1_Safety3_1 AT %I550.2 : Bool;
   S2_R1_Safety4_1 AT %I550.3 : Bool;
   S2_R1_Safety1_2 AT %I550.4 : Bool;
   S2_R1_Safety2_2 AT %I550.5 : Bool;
   S2_R1_Safety3_2 AT %I550.6 : Bool;
   S2_R1_Safety4_2 AT %I550.7 : Bool;
   S2_R1_Valve_Up AT %Q500.0 : Bool;
   S2_R1_Valve_Down AT %Q500.1 : Bool;
   S2_R1_Sen_Drv_1 AT %I500.0 : Bool;
   S2_R1_Sen_Drv_2 AT %I500.1 : Bool;
   S2_R1_Sen_Drv_3 AT %I500.2 : Bool;
   S2_R1_Sen_Drv_4 AT %I500.3 : Bool;
   S2_R1_Sen_Val1_Up AT %I500.4 : Bool;
   S2_R1_Sen_Val1_Down AT %I500.5 : Bool;
   S2_R1_Sen_Val2_Up AT %I500.6 : Bool;
   S2_R1_Sen_Val2_Down AT %I500.7 : Bool;
   S2_R1_Hyd_Filtr AT %I501.0 : Bool;
   S2_R1_Hyd_Empty AT %I501.1 : Bool;
   SS2_R1_ACK_STO AT %Q150.7 : Bool;
   S2_R1_Hydraulic_Unit AT %Q500.2 : Bool;
END_VAR

VAR_GLOBAL   // PLC tag table "S2_R2"
   S2_R2_Safety1_1 AT %I650.0 : Bool;
   S2_R2_Safety2_1 AT %I650.1 : Bool;
   S2_R2_Safety3_1 AT %I650.2 : Bool;
   S2_R2_Safety4_1 AT %I650.3 : Bool;
   S2_R2_Safety1_2 AT %I650.4 : Bool;
   S2_R2_Safety2_2 AT %I650.5 : Bool;
   S2_R2_Safety3_2 AT %I650.6 : Bool;
   S2_R2_Safety4_2 AT %I650.7 : Bool;
   S2_R2_Valve_Up AT %Q600.0 : Bool;
   S2_R2_Valve_Down AT %Q600.1 : Bool;
   S2_R2_Sen_Drv_1 AT %I600.0 : Bool;
   S2_R2_Sen_Drv_2 AT %I600.1 : Bool;
   S2_R2_Sen_Drv_3 AT %I600.2 : Bool;
   S2_R2_Sen_Drv_4 AT %I600.3 : Bool;
   S2_R2_Sen_Val1_Up AT %I600.4 : Bool;
   S2_R2_Sen_Val1_Down AT %I600.5 : Bool;
   S2_R2_Sen_Val2_Up AT %I600.6 : Bool;
   S2_R2_Sen_Val2_Down AT %I600.7 : Bool;
   S2_R2_Hyd_Filtr AT %I601.0 : Bool;
   S2_R2_Hyd_Empty AT %I601.1 : Bool;
   SS2_R2_ACK_STO AT %Q169.7 : Bool;
   iS2L_Distance_Value AT %IW602 : Int;
   S2_R2_Hydraulic_Unit AT %Q600.2 : Bool;
END_VAR

TYPE "CC_Hmi_IO"
   STRUCT
      CC_RollsUp : Bool;
      CC_RollsDown : Bool;
      CC_ModulesUp : Bool;
      CC_ModulesDown : Bool;
      CC_Wibrating : Bool;
      CC_DriveRollerUp : Bool;
      CC_DriveRollerDown : Bool;
   END_STRUCT;
END_TYPE

TYPE "CS_Sides_Stations"
   STRUCT
      RL_H3_Pos : DInt;
      RR_H3_Pos : DInt;
      RL_Mid_Pos : DInt;
      RR_Mid_Pos : DInt;
      RL_H5_Pos : DInt;
      RR_H5_Pos : DInt;
      Correction : Int;
   END_STRUCT;
END_TYPE

TYPE "PII - JN2200"
   STRUCT
      "Process Data Input - Angle Y / vibration acceleration Peak_max" : Int;
      "Process Data Input - Angle X / effective value of the vibration velocity" : Int;
      "Process Data Input - Diagnosis" : Byte;
      "Process Data Input - OUT1" : Bool;
      "Process Data Input - OUT2" : Bool;
      "Reserved Bit" : Bool;
      "Reserved Bit_1" : Bool;
      "Process Data Input - Vibration measurement" : Bool;
      "Process Data Input - Selftest running" : Bool;
      "Reserved Bit_2" : Bool;
      "Reserved Bit_3" : Bool;
   END_STRUCT;
END_TYPE

TYPE "PII - VDM28-50-R1-IO"
   STRUCT
      "Process Data Input - Distance (16 bit)" : Word;
   END_STRUCT;
END_TYPE

TYPE "Pallet"
   STRUCT
      IsSelected : Bool;
      "Name" : String;
      Station_Current_Position : Array[1..2] of Int;
      Number_Of_Elements : Array[1..4] of Int;
   END_STRUCT;
END_TYPE

TYPE "SEW_MOVIKIT_VelocityDrive_SETPOINTS_V2.1"
   STRUCT
      x_Bit_8_Fault_Reset : Bool;
      x_Bit_9_Reserved : Bool;
      x_Bit_10_Activate_DriveTrain2 : Bool;
      x_Bit_11_Reserved : Bool;
      x_Bit_12_Deactivate_SW_Limit_switches : Bool;
      x_Bit_13_Activate_Output_Stage_Inhibit : Bool;
      x_Bit_14_Activate_StandBy_Mode : Bool;
      x_Bit_15_Heartbeat_IN : Bool;
      x_Bit_0_Enable_Emergency_Stop : Bool;
      x_Bit_1_Enable_Application_Stop : Bool;
      x_Bit_2_Reserved : Bool;
      x_Bit_3_Release_Brake : Bool;
      x_Bit_4_Jog_positive : Bool;
      x_Bit_5_Jog_negative : Bool;
      x_Bit_6_Apply_relative_Position : Bool;
      x_Bit_7_Start_Stop : Bool;
      iSetpoint_Speed : Int;
      iSetpoint_Acceleration : Int;
      iSetpoint_Deceleration : Int;
      wDigital_Outputs : Word;
   END_STRUCT;
END_TYPE

TYPE "Station"
   STRUCT
      SensorA : Bool;
      SensorB : Bool;
      SensorC : Bool;
      SensorD : Bool;
      IsEmpty : Bool;
      IsOccupied : Bool;
      Numer : SInt;
      Row : SInt;
      Column : SInt;
   END_STRUCT;
END_TYPE

TYPE "StationLight"
   STRUCT
      SensorA : Bool;
      SensorB : Bool;
      SensorC : Bool;
      SensorD : Bool;
      IsEmpty : Bool;
      IsOccupied : Bool;
      Numer : SInt;
   END_STRUCT;
END_TYPE

TYPE "typeSqlData"
TITLE = typeSqlData
// structure for SQL data received from SELECT command
   STRUCT
      tdsHeader { ExternalAccessible := 'False'; ExternalVisible := 'False'; ExternalWritable := 'False'} : "LSql_typePacketHeader";
      columnCount { ExternalAccessible := 'False'; ExternalVisible := 'False'; ExternalWritable := 'False'} : UInt;   // number of received columns
      columns { ExternalAccessible := 'False'; ExternalVisible := 'False'; ExternalWritable := 'False'} : Array[0.."LSQL_NUMBER_OF_COLUMNS_MAX"] of "LSql_typeColumn";
      rowDataStart { ExternalAccessible := 'False'; ExternalVisible := 'False'; ExternalWritable := 'False'} : UInt;   // start address byte of rowData in TDS telegram
      rowDataLength { ExternalAccessible := 'False'; ExternalVisible := 'False'; ExternalWritable := 'False'} : UDInt;   // area length of rowData in TDS telegram
      rowCount { ExternalAccessible := 'False'; ExternalVisible := 'False'; ExternalWritable := 'False'} : UDInt;   // number of rows
      rowOverflow { ExternalAccessible := 'False'; ExternalVisible := 'False'; ExternalWritable := 'False'} : Bool;   // true = more rows (RowCount) than available UDT tokenRows
      rows { ExternalAccessible := 'False'; ExternalVisible := 'False'; ExternalWritable := 'False'} : Array[0.."LSQL_NUMBER_OF_ROWS_MAX"] of "typeTokenRow";
      errorToken { ExternalAccessible := 'False'; ExternalVisible := 'False'; ExternalWritable := 'False'} : "LSql_typeErrorToken";
   END_STRUCT;
   // // tdsHeader."type" : type of TDS package (4 = Server Response)
   // // tdsHeader.status : status of the TDS package (1= last package, 0 = more packages follow)
   // // tdsHeader.length : length of the TDS response
   // // tdsHeader.spId : process id of the SQL server
   // // tdsHeader.packetID : id of one message for a paket
   // // tdsHeader.window : not used - should be ignored by user
END_TYPE

TYPE "typeTokenRow"
TITLE = typeTokenRow
// use case specific structure for TDS token row
   STRUCT
      Pressure { ExternalAccessible := 'False'; ExternalVisible := 'False'; ExternalWritable := 'False'} : Int;   // row value for column 'Amount'
      Temperature { ExternalAccessible := 'False'; ExternalVisible := 'False'; ExternalWritable := 'False'} : Int;   // row value for column 'Color'
   END_STRUCT;
END_TYPE

DATA_BLOCK "Global_DB"   // DB16
{ S7_Optimized_Access := 'TRUE' }
// stored: MemoryReserve 100
   VAR
      Auto : Bool;
      Manual : Bool;
      Maintenance : Bool;
      Alarm : Word;
   END_VAR
BEGIN
END_DATA_BLOCK

DATA_BLOCK "HMI_DB"   // DB15
{ S7_Optimized_Access := 'TRUE' }
// stored: MemoryReserve 100
   VAR
      ActiveScreenName : String;
      Tip_MT_Control : Bool;
      Tip_HMI_Control : Bool;
      Tip_Up : Bool;
      Tip_Down : Bool;
      TipMT_Arm_Selection : Int;
      TipMT_Button_Up : Bool;
      TipMT_Button_Down : Bool;
      TipMT_Set_Angle : Int;
      TipMT_Button_Open : Bool;
      TipMT_Button_Close : Bool;
      Safety_ACK : Bool;
      Reset_Drives : Bool;
      Reset_Safety : Bool;
      Reset_Reinicialisation : Bool;
      CNTUp : Bool;
      CNTDown : Bool;
      Heart_Bit : USInt;
   END_VAR
BEGIN
END_DATA_BLOCK

DATA_BLOCK "Pallets_Stations"   // DB11
{ S7_Optimized_Access := 'TRUE' }
// stored: MemoryReserve 100
   VAR RETAIN
      Pallets : Array[1..24] of "Pallet";
   END_VAR
   VAR
      Stations : Array[1..4, 1..12] of "Station";
      Stations_ROW1 : Array[1..12] of "StationLight";
      Stations_ROW2 { S7_SetPoint := 'True'} : Array[1..12] of "StationLight";
      Stations_ROW3 { S7_SetPoint := 'True'} : Array[1..12] of "StationLight";
      Stations_ROW4 { S7_SetPoint := 'True'} : Array[1..12] of "StationLight";
   END_VAR
BEGIN
   Stations[1,1..12].Numer := 1;
   Stations[2,1..12].Numer := 2;
   Stations[3,1..12].Numer := 3;
   Stations[4,1..12].Numer := 4;
   Stations[1,1..12].Row := 1;
   Stations[2,1..12].Row := 2;
   Stations[3,1..12].Row := 3;
   Stations[4,1..12].Row := 4;
   Stations[1,1].Column := 1;
   Stations[1,2].Column := 2;
   Stations[1,3].Column := 3;
   Stations[1,4].Column := 4;
   Stations[1,5].Column := 5;
   Stations[1,6].Column := 6;
   Stations[1,7].Column := 7;
   Stations[1,8].Column := 8;
   Stations[1,9].Column := 9;
   Stations[1,10].Column := 10;
   Stations[1,11].Column := 11;
   Stations[1,12].Column := 12;
   Stations[2,1].Column := 1;
   Stations[2,2].Column := 2;
   Stations[2,3].Column := 3;
   Stations[2,4].Column := 4;
   Stations[2,5].Column := 5;
   Stations[2,6].Column := 6;
   Stations[2,7].Column := 7;
   Stations[2,8].Column := 8;
   Stations[2,9].Column := 9;
   Stations[2,10].Column := 10;
   Stations[2,11].Column := 11;
   Stations[2,12].Column := 12;
   Stations[3,1].Column := 1;
   Stations[3,2].Column := 2;
   Stations[3,3].Column := 3;
   Stations[3,4].Column := 4;
   Stations[3,5].Column := 5;
   Stations[3,6].Column := 6;
   Stations[3,7].Column := 7;
   Stations[3,8].Column := 8;
   Stations[3,9].Column := 9;
   Stations[3,10].Column := 10;
   Stations[3,11].Column := 11;
   Stations[3,12].Column := 12;
   Stations[4,1].Column := 1;
   Stations[4,2].Column := 2;
   Stations[4,3].Column := 3;
   Stations[4,4].Column := 4;
   Stations[4,5].Column := 5;
   Stations[4,6].Column := 6;
   Stations[4,7].Column := 7;
   Stations[4,8].Column := 8;
   Stations[4,9].Column := 9;
   Stations[4,10].Column := 10;
   Stations[4,11].Column := 11;
   Stations[4,12].Column := 12;
   Stations_ROW1[1].Numer := 35;
   Stations_ROW1[2].Numer := 34;
   Stations_ROW1[3].Numer := 33;
   Stations_ROW1[4].Numer := 32;
   Stations_ROW1[5].Numer := 31;
   Stations_ROW1[6].Numer := 30;
   Stations_ROW1[7].Numer := 29;
   Stations_ROW1[8].Numer := 28;
   Stations_ROW1[9].Numer := 27;
   Stations_ROW1[10].Numer := 26;
   Stations_ROW1[11].Numer := 25;
   Stations_ROW2[1].Numer := 02;
   Stations_ROW2[2].Numer := 1;
   Stations_ROW2[3].Numer := 38;
   Stations_ROW2[4].Numer := 36;
   Stations_ROW2[5].Numer := 37;
   Stations_ROW2[6].Numer := 18;
   Stations_ROW2[7].Numer := 19;
   Stations_ROW2[8].Numer := 20;
   Stations_ROW2[9].Numer := 21;
   Stations_ROW2[10].Numer := 22;
   Stations_ROW2[11].Numer := 23;
   Stations_ROW2[12].Numer := 24;
   Stations_ROW3[1].Numer := 3;
   Stations_ROW3[11].Numer := 17;
   Stations_ROW4[1].Numer := 4;
   Stations_ROW4[2].Numer := 5;
   Stations_ROW4[3].Numer := 6;
   Stations_ROW4[4].Numer := 7;
   Stations_ROW4[5].Numer := 8;
   Stations_ROW4[6].Numer := 9;
   Stations_ROW4[7].Numer := 10;
   Stations_ROW4[8].Numer := 11;
   Stations_ROW4[9].Numer := 12;
   Stations_ROW4[10].Numer := 13;
   Stations_ROW4[11].Numer := 14;
END_DATA_BLOCK

DATA_BLOCK "CS_MOVIKIT"   // DB28
{ S7_Optimized_Access := 'TRUE' }
// stored: MemoryReserve 100
   VAR
      CS_RL_PI : "SEW_MOVIKIT_VelocityDrive_STATUS_V2.1";
      CS_RL_PO : "SEW_MOVIKIT_VelocityDrive_SETPOINTS_V2.1";
      CS_RP_PI : "SEW_MOVIKIT_VelocityDrive_STATUS_V2.1";
      CS_RP_PO : "SEW_MOVIKIT_VelocityDrive_SETPOINTS_V2.1";
      CS_M1_PI : "SEW_MOVIKIT_VelocityDrive_STATUS_V2.1";
      CS_M1_PO : "SEW_MOVIKIT_VelocityDrive_SETPOINTS_V2.1";
      CS_M2_PI : "SEW_MOVIKIT_VelocityDrive_STATUS_V2.1";
      CS_M2_PO : "SEW_MOVIKIT_VelocityDrive_SETPOINTS_V2.1";
   END_VAR
BEGIN
END_DATA_BLOCK

DATA_BLOCK "CenstralShifter_Diag"   // DB43
{ S7_Optimized_Access := 'TRUE' }
// stored: MemoryReserve 100
   VAR
      Error_num_CS_PL : DInt;
      Error_num_CS_PP : DInt;
      Error_num_CS_TL : DInt;
      Error_num_CS_TP : DInt;
   END_VAR
BEGIN
END_DATA_BLOCK

DATA_BLOCK "EncoderTel81"   // DB44
{ S7_Optimized_Access := 'FALSE' }
   VAR
      Tel81 { S7_SetPoint := 'True'} : PD_TEL81;
   END_VAR
BEGIN
END_DATA_BLOCK

DATA_BLOCK "HMI_Central_Shifter"   // DB32
{ S7_Optimized_Access := 'TRUE' }
// stored: MemoryReserve 100
   VAR
      CS_PP_Reset : Bool;
      CS_PL_Reset : Bool;
      CS_TP_Reset : Bool;
      CS_TL_Reset : Bool;
      CS_Virtual_Reset : Bool;
      CS_Reset : Bool;
      CS_Homing : Bool;
      CS_PP_Power : Bool;
      CS_PL_Power : Bool;
      CS_TP_Power : Bool;
      CS_TL_Power : Bool;
      CS_Virtual_Power : Bool;
      CS_Power : Bool;
      CS_Gear_In : Bool;
      CS_Destination_Pos : Int := 7;
      CS_Drive_To_Des : Bool;
      CS_RL_Hydraulic_Up : Bool;
      CS_RL_Hydraulic_Down : Bool;
      CS_RP_Hydraulic_Up : Bool;
      CS_RP_Hydraulic_Down : Bool;
      CS_RL_Go_Forward : Bool;
      CS_RP_Go_Forward : Bool;
      CS_RP_Go_Backward : Bool;
      CS_RL_Go_Backward : Bool;
      CS_RL_RP_Reset : Bool;
      CS_Sides_Go_Up : Bool;
      CS_Sides_Go_Down : Bool;
      CS_Sides_Go_Mid : Bool;
      CS_Auto : Bool;
      CS_Side_Pos_Up : DInt;
      CS_Side_Pos_Mid : DInt;
      CS_Side_Pos_Down : DInt;
      CS_Pallet_Left_Move : Bool;
      CS_Pallet_Right_Move : Bool;
      CS_Pallet_Centering : Bool;
      CS_Go_Left : Bool;
      CS_Go_Right : Bool;
      CS_Auto_Hyd_Up : Bool;
      CS_Auto_Hyd_Down : Bool;
      CS_Reset_Hydro : Bool;
      CS_Auto_Pos_Start : Int;
      CS_Auto_Pos_End : Int;
      CS_Permission_Auto : Bool;
      CS_Status_Auto_Go_to_Des : SInt;
      Alarms : Word;   // PP/PL/TP/TL Power, GearIN, MoveVirtual
   END_VAR
BEGIN
END_DATA_BLOCK

DATA_BLOCK "DB_CC_HMI"   // DB100
{ S7_Optimized_Access := 'TRUE' }
// stored: AutoNumber false, MemoryReserve 100
   VAR
      Safety_ACK : Bool;
      Reset_Drives : Bool;
      Reset_Safety : Bool;
      Error_Status : Bool;
      CC_ST23_RollsUp : Bool;
      CC_ST23_RollsDown : Bool;
      CC_ST23_ModulesUp : Bool;
      CC_ST23_ModulesDown : Bool;
      CC_ST23_Wibrating : Bool;
      CC_ST23_DriveRollerUp : Bool;
      CC_ST23_DriveRollerDown : Bool;
      CC_ST23_WibratingAuto : Bool;
      CC_ST23_UnlockPallete : Bool;
      CC_ST24_RollsUp : Bool;
      CC_ST24_RollsDown : Bool;
      CC_ST24_ModulesUp : Bool;
      CC_ST24_ModulesDown : Bool;
      CC_ST24_Wibrating : Bool;
      CC_ST24_DriveRollerUp : Bool;
      CC_ST24_DriveRollerDown : Bool;
      CC_ST24_WibratingAuto : Bool;
      CC_ST24_UnlockPallete : Bool;
      CC_ST25_RollsUp : Bool;
      CC_ST25_RollsDown : Bool;
      CC_ST25_ModulesUp : Bool;
      CC_ST25_ModulesDown : Bool;
      CC_ST25_Wibrating : Bool;
      CC_ST25_DriveRollerUp : Bool;
      CC_ST25_DriveRollerDown : Bool;
      CC_ST25_WibratingAuto : Bool;
      CC_ST25_UnlockPallete : Bool;
   END_VAR
BEGIN
END_DATA_BLOCK

DATA_BLOCK "HMI_Pallets"   // DB24
{ S7_Optimized_Access := 'TRUE' }
// stored: MemoryReserve 100
   VAR
      Reset_Drivers : Bool;
      Row : Int;
      Station_Row4 : Int;
      Station_Row2 : Int;
      Station_Row1 : Int;
      Run_Command_left_ROW1 : Array[1..12] of Bool;
      Run_Command_left_ROW2 : Array[1..12] of Bool;
      Run_Command_left_ROW3 : Array[1..12] of Bool;
      Run_Command_left_ROW4 : Array[1..12] of Bool;
      Run_Command_right_ROW1 : Array[1..12] of Bool;
      Run_Command_right_ROW2 : Array[1..12] of Bool;
      Run_Command_right_ROW3 : Array[1..12] of Bool;
      Run_Command_right_ROW4 : Array[1..12] of Bool;
      Run_Status_left_ROW1 : Array[1..12] of Bool;
      Run_Status_left_ROW2 : Array[1..12] of Bool;
      Run_Status_left_ROW3 : Array[1..12] of Bool;
      Run_Status_left_ROW4 : Array[1..12] of Bool;
      Run_Status_right_ROW1 : Array[1..12] of Bool;
      Run_Status_right_ROW2 : Array[1..12] of Bool;
      Run_Status_right_ROW3 : Array[1..12] of Bool;
      Run_Status_right_ROW4 : Array[1..12] of Bool;
      Number_Of_Pallet : SInt;
      Stop_Driver_Button1 : DWord;
      Stop_Driver_HMI1 : DWord;
      Stop_Driver_Button2 : DWord;
      Stop_Driver_HMI2 : DWord;
      Stop_Driver_Status : Bool;
      Drive_Error_Status : Bool;
      Command_Run_W1 : Bool;
      Command_Run_W2 : Bool;
      Command_Run_W4 : Bool;
      Reset_Station_Block_Request : Bool;
      Station_Block_Request_ROW1 : Array[1..12] of Bool;
      Station_Block_Request_ROW2 : Array[1..12] of Bool;
      Station_Block_Request_ROW3 : Array[1..12] of Bool;
      Station_Block_Request_ROW4 : Array[1..12] of Bool;
      Any_Station_Block_ACTIVE : Bool;
      Centering_Alarms : DWord;   // 1-7 -> ROW2, 11-17->ROW4
   END_VAR
BEGIN
END_DATA_BLOCK

DATA_BLOCK "Station_MOVIKIT"   // DB23
{ S7_Optimized_Access := 'TRUE' }
// stored: MemoryReserve 100
   VAR
      MStNONE_PI : "SEW_MOVIKIT_VelocityDrive_STATUS_V2.1";
      MStNONE_PO : "SEW_MOVIKIT_VelocityDrive_SETPOINTS_V2.1";
      MSt1_PI : "SEW_MOVIKIT_VelocityDrive_STATUS_V2.1";
      MSt1_PO : "SEW_MOVIKIT_VelocityDrive_SETPOINTS_V2.1";
      MSt1a_PI : "SEW_MOVIKIT_VelocityDrive_STATUS_V2.1";
      MSt1a_PO : "SEW_MOVIKIT_VelocityDrive_SETPOINTS_V2.1";
      MSt4a_PI : "SEW_MOVIKIT_VelocityDrive_STATUS_V2.1";
      MSt4a_PO : "SEW_MOVIKIT_VelocityDrive_SETPOINTS_V2.1";
      MSt4b_PI : "SEW_MOVIKIT_VelocityDrive_STATUS_V2.1";
      MSt4b_PO : "SEW_MOVIKIT_VelocityDrive_SETPOINTS_V2.1";
      MSt5_PI : "SEW_MOVIKIT_VelocityDrive_STATUS_V2.1";
      MSt5_PO : "SEW_MOVIKIT_VelocityDrive_SETPOINTS_V2.1";
      MSt6a_PI : "SEW_MOVIKIT_VelocityDrive_STATUS_V2.1";
      MSt6a_PO : "SEW_MOVIKIT_VelocityDrive_SETPOINTS_V2.1";
      MSt6b_PI : "SEW_MOVIKIT_VelocityDrive_STATUS_V2.1";
      MSt6b_PO : "SEW_MOVIKIT_VelocityDrive_SETPOINTS_V2.1";
      MSt7_PI : "SEW_MOVIKIT_VelocityDrive_STATUS_V2.1";
      MSt7_PO : "SEW_MOVIKIT_VelocityDrive_SETPOINTS_V2.1";
      MSt8_PI : "SEW_MOVIKIT_VelocityDrive_STATUS_V2.1";
      MSt8_PO : "SEW_MOVIKIT_VelocityDrive_SETPOINTS_V2.1";
      MSt9a_PI : "SEW_MOVIKIT_VelocityDrive_STATUS_V2.1";
      MSt9a_PO : "SEW_MOVIKIT_VelocityDrive_SETPOINTS_V2.1";
      MSt9b_PI : "SEW_MOVIKIT_VelocityDrive_STATUS_V2.1";
      MSt9b_PO : "SEW_MOVIKIT_VelocityDrive_SETPOINTS_V2.1";
      MSt10_PI : "SEW_MOVIKIT_VelocityDrive_STATUS_V2.1";
      MSt10_PO : "SEW_MOVIKIT_VelocityDrive_SETPOINTS_V2.1";
      MSt11_PI : "SEW_MOVIKIT_VelocityDrive_STATUS_V2.1";
      MSt11_PO : "SEW_MOVIKIT_VelocityDrive_SETPOINTS_V2.1";
      MSt12a_PI : "SEW_MOVIKIT_VelocityDrive_STATUS_V2.1";
      MSt12a_PO : "SEW_MOVIKIT_VelocityDrive_SETPOINTS_V2.1";
      MSt12b_PI : "SEW_MOVIKIT_VelocityDrive_STATUS_V2.1";
      MSt12b_PO : "SEW_MOVIKIT_VelocityDrive_SETPOINTS_V2.1";
      MSt13_PI : "SEW_MOVIKIT_VelocityDrive_STATUS_V2.1";
      MSt13_PO : "SEW_MOVIKIT_VelocityDrive_SETPOINTS_V2.1";
      MSt14_PI : "SEW_MOVIKIT_VelocityDrive_STATUS_V2.1";
      MSt14_PO : "SEW_MOVIKIT_VelocityDrive_SETPOINTS_V2.1";
      MSt17_PI : "SEW_MOVIKIT_VelocityDrive_STATUS_V2.1";
      MSt17_PO : "SEW_MOVIKIT_VelocityDrive_SETPOINTS_V2.1";
      MSt18_PI : "SEW_MOVIKIT_VelocityDrive_STATUS_V2.1";
      MSt18_PO : "SEW_MOVIKIT_VelocityDrive_SETPOINTS_V2.1";
      MSt19a_PI : "SEW_MOVIKIT_VelocityDrive_STATUS_V2.1";
      MSt19a_PO : "SEW_MOVIKIT_VelocityDrive_SETPOINTS_V2.1";
      MSt19b_PI : "SEW_MOVIKIT_VelocityDrive_STATUS_V2.1";
      MSt19b_PO : "SEW_MOVIKIT_VelocityDrive_SETPOINTS_V2.1";
      MSt20_PI : "SEW_MOVIKIT_VelocityDrive_STATUS_V2.1";
      MSt20_PO : "SEW_MOVIKIT_VelocityDrive_SETPOINTS_V2.1";
      MSt21_PI : "SEW_MOVIKIT_VelocityDrive_STATUS_V2.1";
      MSt21_PO : "SEW_MOVIKIT_VelocityDrive_SETPOINTS_V2.1";
      MSt22a_PI : "SEW_MOVIKIT_VelocityDrive_STATUS_V2.1";
      MSt22a_PO : "SEW_MOVIKIT_VelocityDrive_SETPOINTS_V2.1";
      MSt22b_PI : "SEW_MOVIKIT_VelocityDrive_STATUS_V2.1";
      MSt22b_PO : "SEW_MOVIKIT_VelocityDrive_SETPOINTS_V2.1";
      MSt23a_PI : "SEW_MOVIKIT_VelocityDrive_STATUS_V2.1";
      MSt23a_PO : "SEW_MOVIKIT_VelocityDrive_SETPOINTS_V2.1";
      MSt23b_PI : "SEW_MOVIKIT_VelocityDrive_STATUS_V2.1";
      MSt23b_PO : "SEW_MOVIKIT_VelocityDrive_SETPOINTS_V2.1";
      MSt24a_PI : "SEW_MOVIKIT_VelocityDrive_STATUS_V2.1";
      MSt24a_PO : "SEW_MOVIKIT_VelocityDrive_SETPOINTS_V2.1";
      MSt24b_PI : "SEW_MOVIKIT_VelocityDrive_STATUS_V2.1";
      MSt24b_PO : "SEW_MOVIKIT_VelocityDrive_SETPOINTS_V2.1";
      MSt25a_PI : "SEW_MOVIKIT_VelocityDrive_STATUS_V2.1";
      MSt25a_PO : "SEW_MOVIKIT_VelocityDrive_SETPOINTS_V2.1";
      MSt25b_PI : "SEW_MOVIKIT_VelocityDrive_STATUS_V2.1";
      MSt25b_PO : "SEW_MOVIKIT_VelocityDrive_SETPOINTS_V2.1";
      MSt26_PI : "SEW_MOVIKIT_VelocityDrive_STATUS_V2.1";
      MSt26_PO : "SEW_MOVIKIT_VelocityDrive_SETPOINTS_V2.1";
      MSt27a_PI : "SEW_MOVIKIT_VelocityDrive_STATUS_V2.1";
      MSt27a_PO : "SEW_MOVIKIT_VelocityDrive_SETPOINTS_V2.1";
      MSt27b_PI : "SEW_MOVIKIT_VelocityDrive_STATUS_V2.1";
      MSt27b_PO : "SEW_MOVIKIT_VelocityDrive_SETPOINTS_V2.1";
      MSt28_PI : "SEW_MOVIKIT_VelocityDrive_STATUS_V2.1";
      MSt28_PO : "SEW_MOVIKIT_VelocityDrive_SETPOINTS_V2.1";
      MSt29_PI : "SEW_MOVIKIT_VelocityDrive_STATUS_V2.1";
      MSt29_PO : "SEW_MOVIKIT_VelocityDrive_SETPOINTS_V2.1";
      MSt30b_PI : "SEW_MOVIKIT_VelocityDrive_STATUS_V2.1";
      MSt30b_PO : "SEW_MOVIKIT_VelocityDrive_SETPOINTS_V2.1";
      MSt30a_PI : "SEW_MOVIKIT_VelocityDrive_STATUS_V2.1";
      MSt30a_PO : "SEW_MOVIKIT_VelocityDrive_SETPOINTS_V2.1";
      MSt31_PI : "SEW_MOVIKIT_VelocityDrive_STATUS_V2.1";
      MSt31_PO : "SEW_MOVIKIT_VelocityDrive_SETPOINTS_V2.1";
      MSt32_PI : "SEW_MOVIKIT_VelocityDrive_STATUS_V2.1";
      MSt32_PO : "SEW_MOVIKIT_VelocityDrive_SETPOINTS_V2.1";
      MSt33a_PI : "SEW_MOVIKIT_VelocityDrive_STATUS_V2.1";
      MSt33a_PO : "SEW_MOVIKIT_VelocityDrive_SETPOINTS_V2.1";
      MSt33b_PI : "SEW_MOVIKIT_VelocityDrive_STATUS_V2.1";
      MSt33b_PO : "SEW_MOVIKIT_VelocityDrive_SETPOINTS_V2.1";
      MSt34_PI : "SEW_MOVIKIT_VelocityDrive_STATUS_V2.1";
      MSt34_PO : "SEW_MOVIKIT_VelocityDrive_SETPOINTS_V2.1";
      MSt35_PI : "SEW_MOVIKIT_VelocityDrive_STATUS_V2.1";
      MSt35_PO : "SEW_MOVIKIT_VelocityDrive_SETPOINTS_V2.1";
      MSt36a_PI : "SEW_MOVIKIT_VelocityDrive_STATUS_V2.1";
      MSt36a_PO : "SEW_MOVIKIT_VelocityDrive_SETPOINTS_V2.1";
      MSt36b_PI : "SEW_MOVIKIT_VelocityDrive_STATUS_V2.1";
      MSt36b_PO : "SEW_MOVIKIT_VelocityDrive_SETPOINTS_V2.1";
      MSt37_PI : "SEW_MOVIKIT_VelocityDrive_STATUS_V2.1";
      MSt37_PO : "SEW_MOVIKIT_VelocityDrive_SETPOINTS_V2.1";
      MSt38_PI : "SEW_MOVIKIT_VelocityDrive_STATUS_V2.1";
      MSt38_PO : "SEW_MOVIKIT_VelocityDrive_SETPOINTS_V2.1";
   END_VAR
BEGIN
   MStNONE_PI.x_Bit_0_Ready := 1;
END_DATA_BLOCK

DATA_BLOCK "Data_From_Safety"   // DB21
{ S7_Optimized_Access := 'TRUE' }
// stored: MemoryReserve 100
   VAR
      Safety_Active : Bool;
      Safety_SS1 : Bool;
      Safety_SS2 : Bool;
      SS1_R1_1 : Bool;
      SS1_R1_2 : Bool;
      SS1_R2_1 : Bool;
      SS1_R2_2 : Bool;
      SS2_R1_1 : Bool;
      SS2_R1_2 : Bool;
      SS2_R2_1 : Bool;
      SS2_R2_2 : Bool;
      Estops : Array[0..14] of Bool;
   END_VAR
BEGIN
END_DATA_BLOCK

DATA_BLOCK "Data_To_Safety"   // DB20
{ S7_Optimized_Access := 'TRUE' }
// stored: MemoryReserve 100
   VAR
      Main_Valve_Arms : Bool;
      Main_Valve_Clamps : Bool;
      Tip_Hydraulic_Unit : Bool;
      Reset_ESTOPS : Bool;
      Reset_REI : Bool;
      Main_Valve_HydRolls : Bool;
   END_VAR
BEGIN
END_DATA_BLOCK

DATA_BLOCK "Tippler_HMI"   // DB401
{ S7_Optimized_Access := 'TRUE' }
// stored: AutoNumber false, MemoryReserve 100
   VAR
      MT_Control : Bool;
      HMI_Control : Bool;
      Up : Bool;
      Down : Bool;
      MT_Arm_Selection : Int;
      Button_Up : Bool;
      Button_Down : Bool;
      Set_Angle : Int;
      MT_Button_Open : Bool;
      MT_Button_Close : Bool;
      MT_Button_Up : Bool;
      MT_Button_Down : Bool;
      Kip1_UP_maint : Bool;
      Kip1_Down_maint : Bool;
      Kip2_UP_maint : Bool;
      Kip2_Down_maint : Bool;
      Kip_Both_Up : Bool;
      Kip_Both_Down : Bool;
   END_VAR
BEGIN
END_DATA_BLOCK

DATA_BLOCK "SqlCommands"   // DB3
TITLE = SqlCommands
{ S7_Optimized_Access := 'TRUE' }
AUTHOR : SIEMENS SUP Applications
VERSION : 1.1
// DB for holding the command strings for a Tabular Data Stream command to a SQL database
// stored: MemoryReserve 0
   VAR
      currentSqlCommand { ExternalAccessible := 'False'; ExternalVisible := 'False'; ExternalWritable := 'False'} : USInt := 6;   // index of current SQL command to be executed (zero-based)
      sqlCommands { ExternalAccessible := 'False'; ExternalVisible := 'False'; ExternalWritable := 'False'} : Array[0..25] of String;   // array of SQL command strings
   END_VAR
BEGIN
   sqlCommands[0] := 'insert into PLCDATA_1 values (7,8, 9)';
   sqlCommands[1] := 'Update PLCDATA_1 set IntegerValue1 = 7, IntegerValue2 = 7, IntegerValue3 = 7 where IntegerValue2 = 7';
   sqlCommands[2] := 'Select IntegerValue1 from PLCDATA_1';
   sqlCommands[3] := 'Select Fruit from PLCDATA_2 where Amount != 0';
   sqlCommands[4] := 'Select Fruit from PLCDATA_2 where color = $'red$'';
   sqlCommands[5] := 'insert into PLCDATA_3 values (7, $'2020-01-01 10:23:24.125$')';
   sqlCommands[6] := 'SELECT TOP (3) * FROM PLCDATA ORDER BY Temperature';
   sqlCommands[7] := 'execute myProcedureIn @input1=30, @input2=6, @input3=84';
   sqlCommands[8] := 'execute myProcedureSelect';
   sqlCommands[9] := 'declare @myout1 char(30),  @myout2 int execute myProcedureInOut @in1=$'pear$', @in2=$'yellow$', @in3=3, @out1=@myout1 OUTPUT, @out2=@myout2 OUTPUT select @myout1 as $'myOut1$', @myOut2 as $'myOut2$'';
   sqlCommands[10] := 'INSERT INTO [dbo].[errors] ([Text]) VALUES ($'remotetest$')';
   sqlCommands[11] := 'SELECT TOP (10) ValueReal1, ValueReal2, ValueReal3, ValueReal4, ValueReal5, ValueReal6, ValueReal7, ValueReal8, ValueReal9 FROM TestJulian';
   sqlCommands[12] := 'SELECT * FROM KompressionLog ORDER BY StentNr';
   sqlCommands[13] := 'execute SelectProc1';
   sqlCommands[14] := 'insert into TestDateTime values ($'01.01.1990 12:00:00$')';
   sqlCommands[15] := 'exec SetDateTime @Input1 = $'07.30.1990 12:00:00$'';
   sqlCommands[16] := 'SELECT TOP (100) MesId, MesId2, MesId3 FROM TestJulian';
   sqlCommands[17] := 'SELECT TOP (1) DateTime FROM TestDateTime';
   sqlCommands[18] := 'SELECT TOP 2 * FROM FunctionTest ORDER BY ID';
   sqlCommands[19] := 'INSERT INTO [dbo].[FunctionTest] DEFAULT VALUES';
   sqlCommands[20] := 'use [SQLFromPLC] declare @myout1 bit  execute  NachtragDatensaetze @inDateiPfad= $'C:\Program Files\Microsoft SQL Server\MSSQL14.SQLEXPRESS\MSSQL\DATA\iO.csv$', @outDone=@myout1 OUTPUT select @myout1 as $'myOut1$'';
   sqlCommands[21] := 'UPDATE [dbo].[KompressionLog] SET LotNummer = $'Test234$' WHERE KammerId = $'3$'';
END_DATA_BLOCK

DATA_BLOCK "SqlConfig"   // DB7
TITLE = SqlConfig
{ S7_Optimized_Access := 'TRUE' }
AUTHOR : SIEMENS SUP Applications
VERSION : 1.1
// DB for providing the connection settings for a Tabuar Data Stream to a SQL database
// stored: MemoryReserve 100
   VAR
      connectionSettings { ExternalAccessible := 'False'; ExternalVisible := 'False'; ExternalWritable := 'False'} : "LSql_typeConnectionSettings";
      enableLSql { ExternalAccessible := 'False'; ExternalVisible := 'False'; ExternalWritable := 'False'} : Bool;   // enables LSql block (starts connection and login, waits for execute commands)
      diagnostics { ExternalWritable := 'False'} : "LSql_typeDiagnostics";
      executeSqlCommand { ExternalAccessible := 'False'; ExternalVisible := 'False'; ExternalWritable := 'False'} : Bool;   // trigger to execute a single sql command. EnableLSql must be true before triggering
   END_VAR
BEGIN
   connectionSettings.interfaceSettings.InterfaceId := 64;
   connectionSettings.interfaceSettings.ID := 16#10;
   connectionSettings.interfaceSettings.ActiveEstablished := true;
   connectionSettings.interfaceSettings.RemoteAddress.ADDR[1] := 10;
   connectionSettings.interfaceSettings.RemoteAddress.ADDR[2..3] := 30;
   connectionSettings.interfaceSettings.RemoteAddress.ADDR[4] := 222;
   connectionSettings.interfaceSettings.RemotePort := 1433;
   connectionSettings.loginInformation.userName := 'SQL_S71500';
   connectionSettings.loginInformation.password := 'SQL_S71500';
   connectionSettings.loginInformation.serverName := 'SQLEXPRESS';
   connectionSettings.loginInformation.databaseName := 'S71500SQLDB';
END_DATA_BLOCK

DATA_BLOCK "SqlData"   // DB5
TITLE = SqlData
{ S7_Optimized_Access := 'TRUE' }
AUTHOR : SIEMENS SUP Applications
VERSION : 3.0
// DB for holding the strucutured data received from a Tabular Data Stream SELECT response
// stored: MemoryReserve 0
   VAR
      data { ExternalAccessible := 'False'; ExternalVisible := 'False'; ExternalWritable := 'False'} : "typeSqlData";
   END_VAR
BEGIN
END_DATA_BLOCK

DATA_BLOCK "SqlTdsReceive"   // DB8
TITLE = SqlTdsReceive
{ S7_Optimized_Access := 'TRUE'; DB_Accessible_From_OPC_UA := 'FALSE' }
AUTHOR : SIEMENS SUP Applications
VERSION : 3.0
// DB for holding the received data array of byte from a Tabular Data Stream (TDS) command to a SQL database
// stored: DBAccessibleFromOPCUA false, MemoryReserve 0
   VAR
      tdsTelegramArrayLength { ExternalAccessible := 'False'; ExternalVisible := 'False'; ExternalWritable := 'False'} : UDInt;   // number of Bytes received by TDS telegram and TRCV input
      tdsTelegramArray { ExternalAccessible := 'False'; ExternalVisible := 'False'; ExternalWritable := 'False'} : Array[0..9999] of Byte;   // array of Bytes of reconstructed TDS telegram
   END_VAR
BEGIN
END_DATA_BLOCK

DATA_BLOCK "HMI_SideShifter_1"   // DB2
{ S7_Optimized_Access := 'TRUE' }
// stored: MemoryReserve 100
   VAR
      SL_Go_Forward : Bool;
      SL_Go_Backward : Bool;
      SL_Velocity : Int;
      SL_Hydraulic_Unit : Bool;
      SL_Actuators_Push : Bool;
      SL_Actuators_Pull : Bool;
      Go_to_ST35 : Bool;
      Go_to_ST02 : Bool;
      Go_to_ST03 : Bool;
      Go_to_ST04 : Bool;
      SR_SL_Hyd_Up : Bool;
      SR_SL_Hyd_Down : Bool;
      SR_Go_Forward : Bool;
      SR_Go_Backward : Bool;
      SR_Velocity : Int;
      SR_Hydraulic_Unit : Bool;
      SR_Actuators_Push : Bool;
      SR_Actuators_Pull : Bool;
      Reset_Drives : Bool;
      Reset_Hydro : Bool;
   END_VAR
   VAR RETAIN
      Homing_SL1 { S7_SetPoint := 'True'} : Int := 1850;
      Homing_SL2 { S7_SetPoint := 'True'} : Int := 7446;
      Homing_SL3 { S7_SetPoint := 'True'} : Int := 13443;
      Homing_SL4 { S7_SetPoint := 'True'} : Int := 19050;
      Homing_SR1 { S7_SetPoint := 'True'} : Int := 1853;
      Homing_SR2 { S7_SetPoint := 'True'} : Int := 7449;
      Homing_SR3 { S7_SetPoint := 'True'} : Int := 13454;
      Homing_SR4 { S7_SetPoint := 'True'} : Int := 19050;
   END_VAR
BEGIN
END_DATA_BLOCK

DATA_BLOCK "HMI_SideShifter_2"   // DB41
{ S7_Optimized_Access := 'TRUE' }
// stored: MemoryReserve 100
   VAR
      SL_Go_Forward : Bool;
      SL_Go_Backward : Bool;
      SL_Velocity : Int;
      SL_Hydraulic_Unit : Bool;
      SL_Actuators_Push : Bool;
      SL_Actuators_Pull : Bool;
      Go_to_ST25 : Bool;
      Go_to_ST24 : Bool;
      Go_to_ST17 : Bool;
      Go_to_ST14 : Bool;
      SR_SL_Hyd_Up : Bool;
      SR_SL_Hyd_Down : Bool;
      SR_Go_Forward : Bool;
      SR_Go_Backward : Bool;
      SR_Velocity : Int;
      SR_Hydraulic_Unit : Bool;
      SR_Actuators_Push : Bool;
      SR_Actuators_Pull : Bool;
      Reset_Drives : Bool;
      Reset_Hydro : Bool;
   END_VAR
   VAR RETAIN
      Homing_SL1 : Int := 1860;
      Homing_SL2 : Int := 7461;
      Homing_SL3 : Int := 13450;
      Homing_SL4 : Int := 19048;
      Homing_SR1 : Int := 1868;
      Homing_SR2 : Int := 7469;
      Homing_SR3 : Int := 13465;
      Homing_SR4 : Int := 19056;
   END_VAR
BEGIN
END_DATA_BLOCK

DATA_BLOCK "Side_MOVIKIT"   // DB18
{ S7_Optimized_Access := 'TRUE' }
// stored: MemoryReserve 0
   VAR
      S2_R1_PI : "SEW_MOVIKIT_VelocityDrive_STATUS_V2.1";
      S2_R1_PO : "SEW_MOVIKIT_VelocityDrive_SETPOINTS_V2.1";
      S2_R2_PI : "SEW_MOVIKIT_VelocityDrive_STATUS_V2.1";
      S2_R2_PO : "SEW_MOVIKIT_VelocityDrive_SETPOINTS_V2.1";
      S2_R1_Communication_OK { S7_SetPoint := 'True'} : Bool;
      S2_R2_Communication_OK { S7_SetPoint := 'True'} : Bool;
      S1_R1_PI : "SEW_MOVIKIT_VelocityDrive_STATUS_V2.1";
      S1_R1_PO : "SEW_MOVIKIT_VelocityDrive_SETPOINTS_V2.1";
      S1_R2_PI : "SEW_MOVIKIT_VelocityDrive_STATUS_V2.1";
      S1_R2_PO : "SEW_MOVIKIT_VelocityDrive_SETPOINTS_V2.1";
      S1_R1_Communication_OK { S7_SetPoint := 'True'} : Bool;
      S1_R2_Communication_OK { S7_SetPoint := 'True'} : Bool;
   END_VAR
BEGIN
END_DATA_BLOCK

ORGANIZATION_BLOCK "Main"   // OB1, LAD, ProgramCycle
TITLE = "Main Program Sweep (Cycle)"
{ S7_Optimized_Access := 'TRUE' }
// stored: SetENOAutomatically false
   VAR_INPUT
      Initial_Call : Bool;   // Initial call of this OB
      Remanence : Bool;   // =True, if remanent data are available
   END_VAR
BEGIN

REGION Network 1: SideShifter2
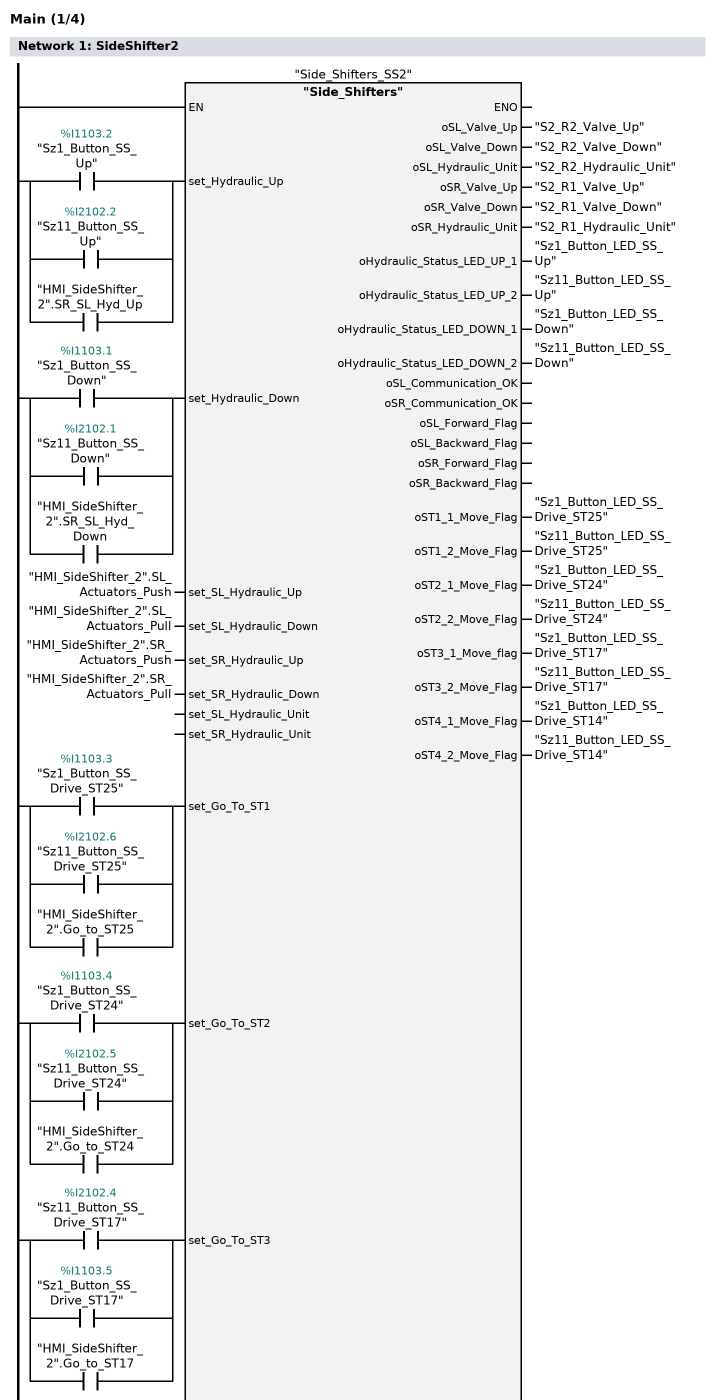
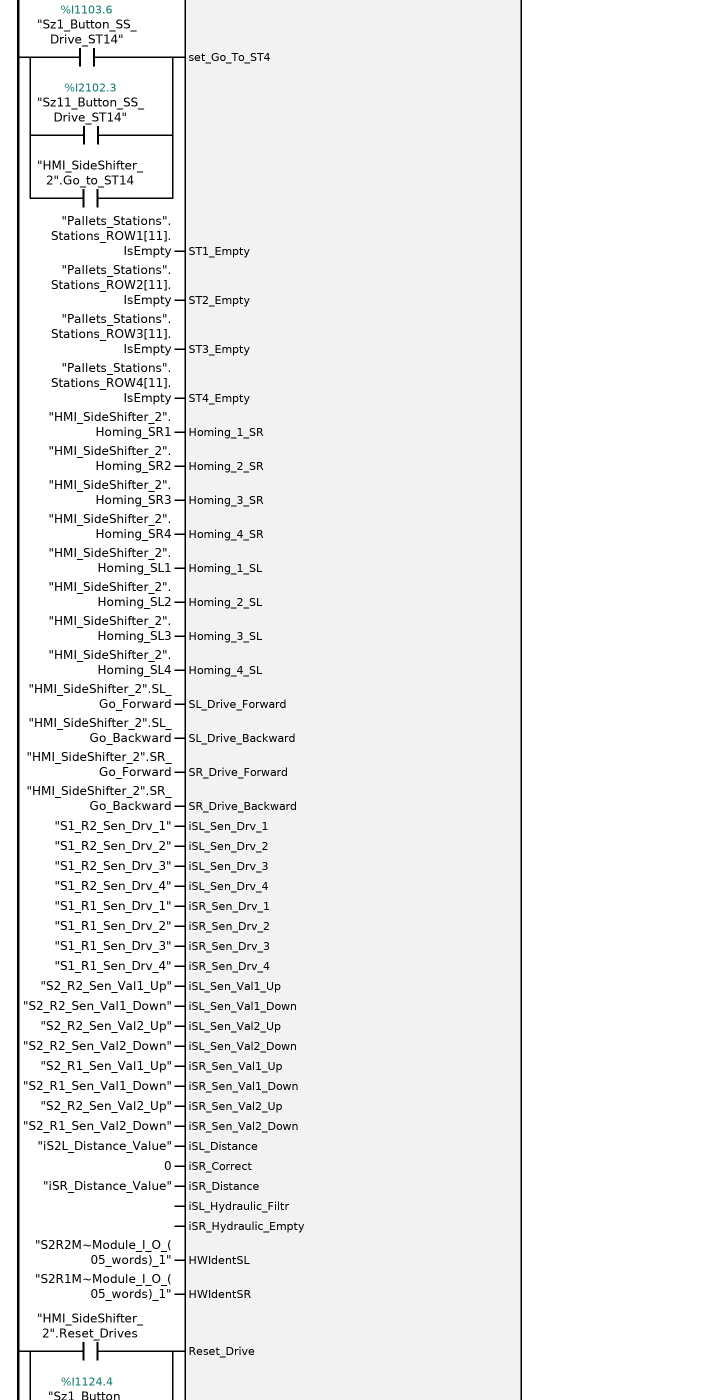
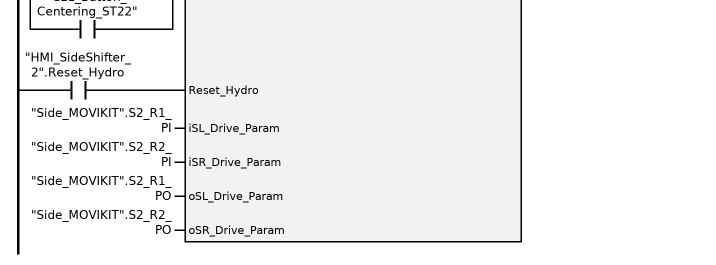
   RUNG wire#powerrail
      "Side_Shifters_SS2"(set_Hydraulic_Up := wire#w1, set_Hydraulic_Down := wire#w2, set_Go_To_ST1 := wire#w3, set_Go_To_ST2 := wire#w4, set_Go_To_ST3 := wire#w5, set_Go_To_ST4 := wire#w6, Reset_Drive := wire#w7, Reset_Hydro := wire#w8, set_SL_Hydraulic_Up := "HMI_SideShifter_2".SL_Actuators_Push, set_SL_Hydraulic_Down := "HMI_SideShifter_2".SL_Actuators_Pull, set_SR_Hydraulic_Up := "HMI_SideShifter_2".SR_Actuators_Push, set_SR_Hydraulic_Down := "HMI_SideShifter_2".SR_Actuators_Pull, set_SL_Hydraulic_Unit :=, set_SR_Hydraulic_Unit :=, ST1_Empty := "Pallets_Stations".Stations_ROW1[11].IsEmpty, ST2_Empty := "Pallets_Stations".Stations_ROW2[11].IsEmpty, ST3_Empty := "Pallets_Stations".Stations_ROW3[11].IsEmpty, ST4_Empty := "Pallets_Stations".Stations_ROW4[11].IsEmpty, Homing_1_SR := "HMI_SideShifter_2".Homing_SR1, Homing_2_SR := "HMI_SideShifter_2".Homing_SR2, Homing_3_SR := "HMI_SideShifter_2".Homing_SR3, Homing_4_SR := "HMI_SideShifter_2".Homing_SR4, Homing_1_SL := "HMI_SideShifter_2".Homing_SL1, Homing_2_SL := "HMI_SideShifter_2".Homing_SL2, Homing_3_SL := "HMI_SideShifter_2".Homing_SL3, Homing_4_SL := "HMI_SideShifter_2".Homing_SL4, SL_Drive_Forward := "HMI_SideShifter_2".SL_Go_Forward, SL_Drive_Backward := "HMI_SideShifter_2".SL_Go_Backward, SR_Drive_Forward := "HMI_SideShifter_2".SR_Go_Forward, SR_Drive_Backward := "HMI_SideShifter_2".SR_Go_Backward, iSL_Sen_Drv_1 := "S1_R2_Sen_Drv_1", iSL_Sen_Drv_2 := "S1_R2_Sen_Drv_2", iSL_Sen_Drv_3 := "S1_R2_Sen_Drv_3", iSL_Sen_Drv_4 := "S1_R2_Sen_Drv_4", iSR_Sen_Drv_1 := "S1_R1_Sen_Drv_1", iSR_Sen_Drv_2 := "S1_R1_Sen_Drv_2", iSR_Sen_Drv_3 := "S1_R1_Sen_Drv_3", iSR_Sen_Drv_4 := "S1_R1_Sen_Drv_4", iSL_Sen_Val1_Up := "S2_R2_Sen_Val1_Up", iSL_Sen_Val1_Down := "S2_R2_Sen_Val1_Down", iSL_Sen_Val2_Up := "S2_R2_Sen_Val2_Up", iSL_Sen_Val2_Down := "S2_R2_Sen_Val2_Down", iSR_Sen_Val1_Up := "S2_R1_Sen_Val1_Up", iSR_Sen_Val1_Down := "S2_R1_Sen_Val1_Down", iSR_Sen_Val2_Up := "S2_R2_Sen_Val2_Up", iSR_Sen_Val2_Down := "S2_R1_Sen_Val2_Down", iSL_Distance := "iS2L_Distance_Value", iSR_Correct := 0, iSR_Distance := "iSR_Distance_Value", iSL_Hydraulic_Filtr :=, iSR_Hydraulic_Empty :=, HWIdentSL := "S2R2M~Module_I_O_(05_words)_1", HWIdentSR := "S2R1M~Module_I_O_(05_words)_1", iSL_Drive_Param := "Side_MOVIKIT".S2_R1_PI, iSR_Drive_Param := "Side_MOVIKIT".S2_R2_PI, oSL_Drive_Param := "Side_MOVIKIT".S2_R1_PO, oSR_Drive_Param := "Side_MOVIKIT".S2_R2_PO, oSL_Valve_Up => "S2_R2_Valve_Up", oSL_Valve_Down => "S2_R2_Valve_Down", oSL_Hydraulic_Unit => "S2_R2_Hydraulic_Unit", oSR_Valve_Up => "S2_R1_Valve_Up", oSR_Valve_Down => "S2_R1_Valve_Down", oSR_Hydraulic_Unit => "S2_R1_Hydraulic_Unit", oHydraulic_Status_LED_UP_1 => "Sz1_Button_LED_SS_Up", oHydraulic_Status_LED_UP_2 => "Sz11_Button_LED_SS_Up", oHydraulic_Status_LED_DOWN_1 => "Sz1_Button_LED_SS_Down", oHydraulic_Status_LED_DOWN_2 => "Sz11_Button_LED_SS_Down", oSL_Communication_OK =>, oSR_Communication_OK =>, oSL_Forward_Flag =>, oSL_Backward_Flag =>, oSR_Forward_Flag =>, oSR_Backward_Flag =>, oST1_1_Move_Flag => "Sz1_Button_LED_SS_Drive_ST25", oST1_2_Move_Flag => "Sz11_Button_LED_SS_Drive_ST25", oST2_1_Move_Flag => "Sz1_Button_LED_SS_Drive_ST24", oST2_2_Move_Flag => "Sz11_Button_LED_SS_Drive_ST24", oST3_1_Move_flag => "Sz1_Button_LED_SS_Drive_ST17", oST3_2_Move_Flag => "Sz11_Button_LED_SS_Drive_ST17", oST4_1_Move_Flag => "Sz1_Button_LED_SS_Drive_ST14", oST4_2_Move_Flag => "Sz11_Button_LED_SS_Drive_ST14")
   END_RUNG
   RUNG wire#powerrail
      Contact( "Sz1_Button_SS_Up" )
   END_RUNG wire#w1
   RUNG wire#powerrail
      Contact( "Sz11_Button_SS_Up" )
   END_RUNG wire#w1
   RUNG wire#powerrail
      Contact( "HMI_SideShifter_2".SR_SL_Hyd_Up )
   END_RUNG wire#w1
   RUNG wire#powerrail
      Contact( "Sz1_Button_SS_Down" )
   END_RUNG wire#w2
   RUNG wire#powerrail
      Contact( "Sz11_Button_SS_Down" )
   END_RUNG wire#w2
   RUNG wire#powerrail
      Contact( "HMI_SideShifter_2".SR_SL_Hyd_Down )
   END_RUNG wire#w2
   RUNG wire#powerrail
      Contact( "Sz1_Button_SS_Drive_ST25" )
   END_RUNG wire#w3
   RUNG wire#powerrail
      Contact( "Sz11_Button_SS_Drive_ST25" )
   END_RUNG wire#w3
   RUNG wire#powerrail
      Contact( "HMI_SideShifter_2".Go_to_ST25 )
   END_RUNG wire#w3
   RUNG wire#powerrail
      Contact( "Sz1_Button_SS_Drive_ST24" )
   END_RUNG wire#w4
   RUNG wire#powerrail
      Contact( "Sz11_Button_SS_Drive_ST24" )
   END_RUNG wire#w4
   RUNG wire#powerrail
      Contact( "HMI_SideShifter_2".Go_to_ST24 )
   END_RUNG wire#w4
   RUNG wire#powerrail
      Contact( "Sz11_Button_SS_Drive_ST17" )
   END_RUNG wire#w5
   RUNG wire#powerrail
      Contact( "Sz1_Button_SS_Drive_ST17" )
   END_RUNG wire#w5
   RUNG wire#powerrail
      Contact( "HMI_SideShifter_2".Go_to_ST17 )
   END_RUNG wire#w5
   RUNG wire#powerrail
      Contact( "Sz1_Button_SS_Drive_ST14" )
   END_RUNG wire#w6
   RUNG wire#powerrail
      Contact( "Sz11_Button_SS_Drive_ST14" )
   END_RUNG wire#w6
   RUNG wire#powerrail
      Contact( "HMI_SideShifter_2".Go_to_ST14 )
   END_RUNG wire#w6
   RUNG wire#powerrail
      Contact( "HMI_SideShifter_2".Reset_Drives )
   END_RUNG wire#w7
   RUNG wire#powerrail
      Contact( "Sz1_Button_Centering_ST22" )
   END_RUNG wire#w7
   RUNG wire#powerrail
      Contact( "HMI_SideShifter_2".Reset_Hydro )
   END_RUNG wire#w8
   // the same network as SCL:
   "Side_Shifters_SS2"(set_Hydraulic_Up := "Sz1_Button_SS_Up" OR "Sz11_Button_SS_Up" OR "HMI_SideShifter_2".SR_SL_Hyd_Up,   // "Side_Shifters"
                       set_Hydraulic_Down := "Sz1_Button_SS_Down" OR "Sz11_Button_SS_Down" OR "HMI_SideShifter_2".SR_SL_Hyd_Down,
                       set_SL_Hydraulic_Up := "HMI_SideShifter_2".SL_Actuators_Push,
                       set_SL_Hydraulic_Down := "HMI_SideShifter_2".SL_Actuators_Pull,
                       set_SR_Hydraulic_Up := "HMI_SideShifter_2".SR_Actuators_Push,
                       set_SR_Hydraulic_Down := "HMI_SideShifter_2".SR_Actuators_Pull,
                       set_Go_To_ST1 := "Sz1_Button_SS_Drive_ST25" OR "Sz11_Button_SS_Drive_ST25" OR "HMI_SideShifter_2".Go_to_ST25,
                       set_Go_To_ST2 := "Sz1_Button_SS_Drive_ST24" OR "Sz11_Button_SS_Drive_ST24" OR "HMI_SideShifter_2".Go_to_ST24,
                       set_Go_To_ST3 := "Sz11_Button_SS_Drive_ST17" OR "Sz1_Button_SS_Drive_ST17" OR "HMI_SideShifter_2".Go_to_ST17,
                       set_Go_To_ST4 := "Sz1_Button_SS_Drive_ST14" OR "Sz11_Button_SS_Drive_ST14" OR "HMI_SideShifter_2".Go_to_ST14,
                       ST1_Empty := "Pallets_Stations".Stations_ROW1[11].IsEmpty,
                       ST2_Empty := "Pallets_Stations".Stations_ROW2[11].IsEmpty,
                       ST3_Empty := "Pallets_Stations".Stations_ROW3[11].IsEmpty,
                       ST4_Empty := "Pallets_Stations".Stations_ROW4[11].IsEmpty,
                       Homing_1_SR := "HMI_SideShifter_2".Homing_SR1,
                       Homing_2_SR := "HMI_SideShifter_2".Homing_SR2,
                       Homing_3_SR := "HMI_SideShifter_2".Homing_SR3,
                       Homing_4_SR := "HMI_SideShifter_2".Homing_SR4,
                       Homing_1_SL := "HMI_SideShifter_2".Homing_SL1,
                       Homing_2_SL := "HMI_SideShifter_2".Homing_SL2,
                       Homing_3_SL := "HMI_SideShifter_2".Homing_SL3,
                       Homing_4_SL := "HMI_SideShifter_2".Homing_SL4,
                       SL_Drive_Forward := "HMI_SideShifter_2".SL_Go_Forward,
                       SL_Drive_Backward := "HMI_SideShifter_2".SL_Go_Backward,
                       SR_Drive_Forward := "HMI_SideShifter_2".SR_Go_Forward,
                       SR_Drive_Backward := "HMI_SideShifter_2".SR_Go_Backward,
                       iSL_Sen_Drv_1 := "S1_R2_Sen_Drv_1",
                       iSL_Sen_Drv_2 := "S1_R2_Sen_Drv_2",
                       iSL_Sen_Drv_3 := "S1_R2_Sen_Drv_3",
                       iSL_Sen_Drv_4 := "S1_R2_Sen_Drv_4",
                       iSR_Sen_Drv_1 := "S1_R1_Sen_Drv_1",
                       iSR_Sen_Drv_2 := "S1_R1_Sen_Drv_2",
                       iSR_Sen_Drv_3 := "S1_R1_Sen_Drv_3",
                       iSR_Sen_Drv_4 := "S1_R1_Sen_Drv_4",
                       iSL_Sen_Val1_Up := "S2_R2_Sen_Val1_Up",
                       iSL_Sen_Val1_Down := "S2_R2_Sen_Val1_Down",
                       iSL_Sen_Val2_Up := "S2_R2_Sen_Val2_Up",
                       iSL_Sen_Val2_Down := "S2_R2_Sen_Val2_Down",
                       iSR_Sen_Val1_Up := "S2_R1_Sen_Val1_Up",
                       iSR_Sen_Val1_Down := "S2_R1_Sen_Val1_Down",
                       iSR_Sen_Val2_Up := "S2_R2_Sen_Val2_Up",
                       iSR_Sen_Val2_Down := "S2_R1_Sen_Val2_Down",
                       iSL_Distance := "iS2L_Distance_Value",
                       iSR_Correct := 0,
                       iSR_Distance := "iSR_Distance_Value",
                       HWIdentSL := "S2R2M~Module_I_O_(05_words)_1",
                       HWIdentSR := "S2R1M~Module_I_O_(05_words)_1",
                       Reset_Drive := "HMI_SideShifter_2".Reset_Drives OR "Sz1_Button_Centering_ST22",
                       Reset_Hydro := "HMI_SideShifter_2".Reset_Hydro,
                       iSL_Drive_Param := "Side_MOVIKIT".S2_R1_PI,
                       iSR_Drive_Param := "Side_MOVIKIT".S2_R2_PI,
                       oSL_Drive_Param := "Side_MOVIKIT".S2_R1_PO,
                       oSR_Drive_Param := "Side_MOVIKIT".S2_R2_PO,
                       oSL_Valve_Up => "S2_R2_Valve_Up",
                       oSL_Valve_Down => "S2_R2_Valve_Down",
                       oSL_Hydraulic_Unit => "S2_R2_Hydraulic_Unit",
                       oSR_Valve_Up => "S2_R1_Valve_Up",
                       oSR_Valve_Down => "S2_R1_Valve_Down",
                       oSR_Hydraulic_Unit => "S2_R1_Hydraulic_Unit",
                       oHydraulic_Status_LED_UP_1 => "Sz1_Button_LED_SS_Up",
                       oHydraulic_Status_LED_UP_2 => "Sz11_Button_LED_SS_Up",
                       oHydraulic_Status_LED_DOWN_1 => "Sz1_Button_LED_SS_Down",
                       oHydraulic_Status_LED_DOWN_2 => "Sz11_Button_LED_SS_Down",
                       oST1_1_Move_Flag => "Sz1_Button_LED_SS_Drive_ST25",
                       oST1_2_Move_Flag => "Sz11_Button_LED_SS_Drive_ST25",
                       oST2_1_Move_Flag => "Sz1_Button_LED_SS_Drive_ST24",
                       oST2_2_Move_Flag => "Sz11_Button_LED_SS_Drive_ST24",
                       oST3_1_Move_flag => "Sz1_Button_LED_SS_Drive_ST17",
                       oST3_2_Move_Flag => "Sz11_Button_LED_SS_Drive_ST17",
                       oST4_1_Move_Flag => "Sz1_Button_LED_SS_Drive_ST14",
                       oST4_2_Move_Flag => "Sz11_Button_LED_SS_Drive_ST14");
END_REGION

REGION Network 2: SideShifter 1
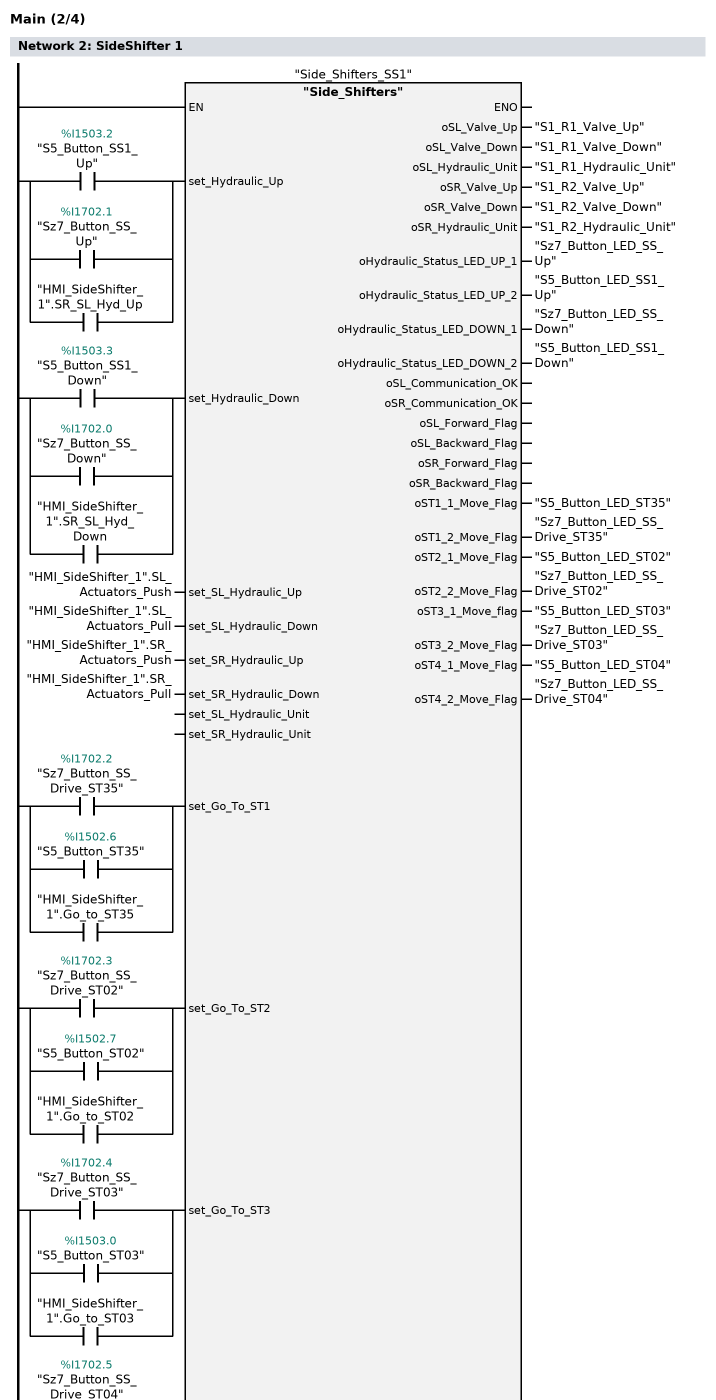
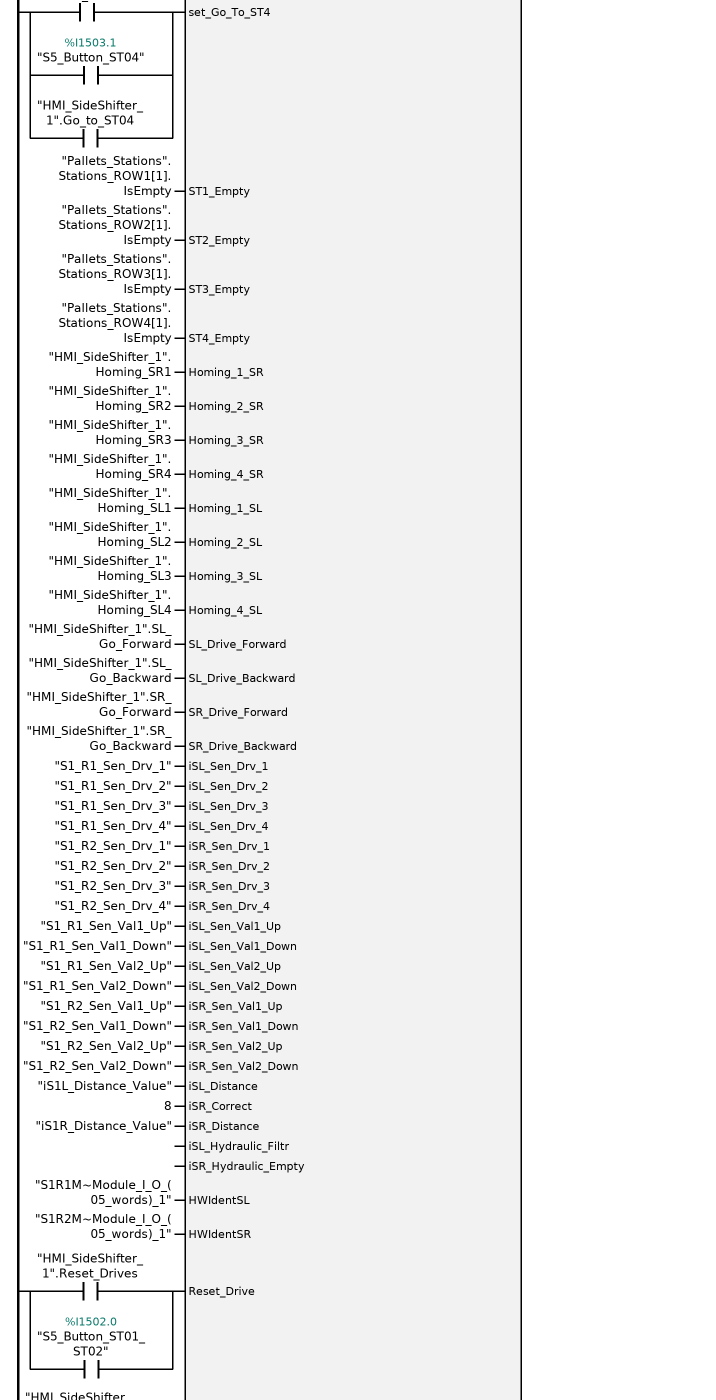
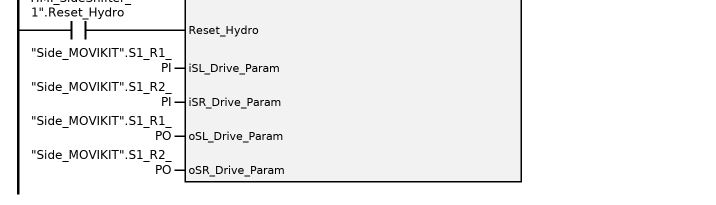
   RUNG wire#powerrail
      "Side_Shifters_SS1"(set_Hydraulic_Up := wire#w1, set_Hydraulic_Down := wire#w2, set_Go_To_ST1 := wire#w3, set_Go_To_ST2 := wire#w4, set_Go_To_ST3 := wire#w5, set_Go_To_ST4 := wire#w6, Reset_Drive := wire#w7, Reset_Hydro := wire#w8, set_SL_Hydraulic_Up := "HMI_SideShifter_1".SL_Actuators_Push, set_SL_Hydraulic_Down := "HMI_SideShifter_1".SL_Actuators_Pull, set_SR_Hydraulic_Up := "HMI_SideShifter_1".SR_Actuators_Push, set_SR_Hydraulic_Down := "HMI_SideShifter_1".SR_Actuators_Pull, set_SL_Hydraulic_Unit :=, set_SR_Hydraulic_Unit :=, ST1_Empty := "Pallets_Stations".Stations_ROW1[1].IsEmpty, ST2_Empty := "Pallets_Stations".Stations_ROW2[1].IsEmpty, ST3_Empty := "Pallets_Stations".Stations_ROW3[1].IsEmpty, ST4_Empty := "Pallets_Stations".Stations_ROW4[1].IsEmpty, Homing_1_SR := "HMI_SideShifter_1".Homing_SR1, Homing_2_SR := "HMI_SideShifter_1".Homing_SR2, Homing_3_SR := "HMI_SideShifter_1".Homing_SR3, Homing_4_SR := "HMI_SideShifter_1".Homing_SR4, Homing_1_SL := "HMI_SideShifter_1".Homing_SL1, Homing_2_SL := "HMI_SideShifter_1".Homing_SL2, Homing_3_SL := "HMI_SideShifter_1".Homing_SL3, Homing_4_SL := "HMI_SideShifter_1".Homing_SL4, SL_Drive_Forward := "HMI_SideShifter_1".SL_Go_Forward, SL_Drive_Backward := "HMI_SideShifter_1".SL_Go_Backward, SR_Drive_Forward := "HMI_SideShifter_1".SR_Go_Forward, SR_Drive_Backward := "HMI_SideShifter_1".SR_Go_Backward, iSL_Sen_Drv_1 := "S1_R1_Sen_Drv_1", iSL_Sen_Drv_2 := "S1_R1_Sen_Drv_2", iSL_Sen_Drv_3 := "S1_R1_Sen_Drv_3", iSL_Sen_Drv_4 := "S1_R1_Sen_Drv_4", iSR_Sen_Drv_1 := "S1_R2_Sen_Drv_1", iSR_Sen_Drv_2 := "S1_R2_Sen_Drv_2", iSR_Sen_Drv_3 := "S1_R2_Sen_Drv_3", iSR_Sen_Drv_4 := "S1_R2_Sen_Drv_4", iSL_Sen_Val1_Up := "S1_R1_Sen_Val1_Up", iSL_Sen_Val1_Down := "S1_R1_Sen_Val1_Down", iSL_Sen_Val2_Up := "S1_R1_Sen_Val2_Up", iSL_Sen_Val2_Down := "S1_R1_Sen_Val2_Down", iSR_Sen_Val1_Up := "S1_R2_Sen_Val1_Up", iSR_Sen_Val1_Down := "S1_R2_Sen_Val1_Down", iSR_Sen_Val2_Up := "S1_R2_Sen_Val2_Up", iSR_Sen_Val2_Down := "S1_R2_Sen_Val2_Down", iSL_Distance := "iS1L_Distance_Value", iSR_Correct := 8, iSR_Distance := "iS1R_Distance_Value", iSL_Hydraulic_Filtr :=, iSR_Hydraulic_Empty :=, HWIdentSL := "S1R1M~Module_I_O_(05_words)_1", HWIdentSR := "S1R2M~Module_I_O_(05_words)_1", iSL_Drive_Param := "Side_MOVIKIT".S1_R1_PI, iSR_Drive_Param := "Side_MOVIKIT".S1_R2_PI, oSL_Drive_Param := "Side_MOVIKIT".S1_R1_PO, oSR_Drive_Param := "Side_MOVIKIT".S1_R2_PO, oSL_Valve_Up => "S1_R1_Valve_Up", oSL_Valve_Down => "S1_R1_Valve_Down", oSL_Hydraulic_Unit => "S1_R1_Hydraulic_Unit", oSR_Valve_Up => "S1_R2_Valve_Up", oSR_Valve_Down => "S1_R2_Valve_Down", oSR_Hydraulic_Unit => "S1_R2_Hydraulic_Unit", oHydraulic_Status_LED_UP_1 => "Sz7_Button_LED_SS_Up", oHydraulic_Status_LED_UP_2 => "S5_Button_LED_SS1_Up", oHydraulic_Status_LED_DOWN_1 => "Sz7_Button_LED_SS_Down", oHydraulic_Status_LED_DOWN_2 => "S5_Button_LED_SS1_Down", oSL_Communication_OK =>, oSR_Communication_OK =>, oSL_Forward_Flag =>, oSL_Backward_Flag =>, oSR_Forward_Flag =>, oSR_Backward_Flag =>, oST1_1_Move_Flag => "S5_Button_LED_ST35", oST1_2_Move_Flag => "Sz7_Button_LED_SS_Drive_ST35", oST2_1_Move_Flag => "S5_Button_LED_ST02", oST2_2_Move_Flag => "Sz7_Button_LED_SS_Drive_ST02", oST3_1_Move_flag => "S5_Button_LED_ST03", oST3_2_Move_Flag => "Sz7_Button_LED_SS_Drive_ST03", oST4_1_Move_Flag => "S5_Button_LED_ST04", oST4_2_Move_Flag => "Sz7_Button_LED_SS_Drive_ST04")
   END_RUNG
   RUNG wire#powerrail
      Contact( "S5_Button_SS1_Up" )
   END_RUNG wire#w1
   RUNG wire#powerrail
      Contact( "Sz7_Button_SS_Up" )
   END_RUNG wire#w1
   RUNG wire#powerrail
      Contact( "HMI_SideShifter_1".SR_SL_Hyd_Up )
   END_RUNG wire#w1
   RUNG wire#powerrail
      Contact( "S5_Button_SS1_Down" )
   END_RUNG wire#w2
   RUNG wire#powerrail
      Contact( "Sz7_Button_SS_Down" )
   END_RUNG wire#w2
   RUNG wire#powerrail
      Contact( "HMI_SideShifter_1".SR_SL_Hyd_Down )
   END_RUNG wire#w2
   RUNG wire#powerrail
      Contact( "Sz7_Button_SS_Drive_ST35" )
   END_RUNG wire#w3
   RUNG wire#powerrail
      Contact( "S5_Button_ST35" )
   END_RUNG wire#w3
   RUNG wire#powerrail
      Contact( "HMI_SideShifter_1".Go_to_ST35 )
   END_RUNG wire#w3
   RUNG wire#powerrail
      Contact( "Sz7_Button_SS_Drive_ST02" )
   END_RUNG wire#w4
   RUNG wire#powerrail
      Contact( "S5_Button_ST02" )
   END_RUNG wire#w4
   RUNG wire#powerrail
      Contact( "HMI_SideShifter_1".Go_to_ST02 )
   END_RUNG wire#w4
   RUNG wire#powerrail
      Contact( "Sz7_Button_SS_Drive_ST03" )
   END_RUNG wire#w5
   RUNG wire#powerrail
      Contact( "S5_Button_ST03" )
   END_RUNG wire#w5
   RUNG wire#powerrail
      Contact( "HMI_SideShifter_1".Go_to_ST03 )
   END_RUNG wire#w5
   RUNG wire#powerrail
      Contact( "Sz7_Button_SS_Drive_ST04" )
   END_RUNG wire#w6
   RUNG wire#powerrail
      Contact( "S5_Button_ST04" )
   END_RUNG wire#w6
   RUNG wire#powerrail
      Contact( "HMI_SideShifter_1".Go_to_ST04 )
   END_RUNG wire#w6
   RUNG wire#powerrail
      Contact( "HMI_SideShifter_1".Reset_Drives )
   END_RUNG wire#w7
   RUNG wire#powerrail
      Contact( "S5_Button_ST01_ST02" )
   END_RUNG wire#w7
   RUNG wire#powerrail
      Contact( "HMI_SideShifter_1".Reset_Hydro )
   END_RUNG wire#w8
   // the same network as SCL:
   "Side_Shifters_SS1"(set_Hydraulic_Up := "S5_Button_SS1_Up" OR "Sz7_Button_SS_Up" OR "HMI_SideShifter_1".SR_SL_Hyd_Up,   // "Side_Shifters"
                       set_Hydraulic_Down := "S5_Button_SS1_Down" OR "Sz7_Button_SS_Down" OR "HMI_SideShifter_1".SR_SL_Hyd_Down,
                       set_SL_Hydraulic_Up := "HMI_SideShifter_1".SL_Actuators_Push,
                       set_SL_Hydraulic_Down := "HMI_SideShifter_1".SL_Actuators_Pull,
                       set_SR_Hydraulic_Up := "HMI_SideShifter_1".SR_Actuators_Push,
                       set_SR_Hydraulic_Down := "HMI_SideShifter_1".SR_Actuators_Pull,
                       set_Go_To_ST1 := "Sz7_Button_SS_Drive_ST35" OR "S5_Button_ST35" OR "HMI_SideShifter_1".Go_to_ST35,
                       set_Go_To_ST2 := "Sz7_Button_SS_Drive_ST02" OR "S5_Button_ST02" OR "HMI_SideShifter_1".Go_to_ST02,
                       set_Go_To_ST3 := "Sz7_Button_SS_Drive_ST03" OR "S5_Button_ST03" OR "HMI_SideShifter_1".Go_to_ST03,
                       set_Go_To_ST4 := "Sz7_Button_SS_Drive_ST04" OR "S5_Button_ST04" OR "HMI_SideShifter_1".Go_to_ST04,
                       ST1_Empty := "Pallets_Stations".Stations_ROW1[1].IsEmpty,
                       ST2_Empty := "Pallets_Stations".Stations_ROW2[1].IsEmpty,
                       ST3_Empty := "Pallets_Stations".Stations_ROW3[1].IsEmpty,
                       ST4_Empty := "Pallets_Stations".Stations_ROW4[1].IsEmpty,
                       Homing_1_SR := "HMI_SideShifter_1".Homing_SR1,
                       Homing_2_SR := "HMI_SideShifter_1".Homing_SR2,
                       Homing_3_SR := "HMI_SideShifter_1".Homing_SR3,
                       Homing_4_SR := "HMI_SideShifter_1".Homing_SR4,
                       Homing_1_SL := "HMI_SideShifter_1".Homing_SL1,
                       Homing_2_SL := "HMI_SideShifter_1".Homing_SL2,
                       Homing_3_SL := "HMI_SideShifter_1".Homing_SL3,
                       Homing_4_SL := "HMI_SideShifter_1".Homing_SL4,
                       SL_Drive_Forward := "HMI_SideShifter_1".SL_Go_Forward,
                       SL_Drive_Backward := "HMI_SideShifter_1".SL_Go_Backward,
                       SR_Drive_Forward := "HMI_SideShifter_1".SR_Go_Forward,
                       SR_Drive_Backward := "HMI_SideShifter_1".SR_Go_Backward,
                       iSL_Sen_Drv_1 := "S1_R1_Sen_Drv_1",
                       iSL_Sen_Drv_2 := "S1_R1_Sen_Drv_2",
                       iSL_Sen_Drv_3 := "S1_R1_Sen_Drv_3",
                       iSL_Sen_Drv_4 := "S1_R1_Sen_Drv_4",
                       iSR_Sen_Drv_1 := "S1_R2_Sen_Drv_1",
                       iSR_Sen_Drv_2 := "S1_R2_Sen_Drv_2",
                       iSR_Sen_Drv_3 := "S1_R2_Sen_Drv_3",
                       iSR_Sen_Drv_4 := "S1_R2_Sen_Drv_4",
                       iSL_Sen_Val1_Up := "S1_R1_Sen_Val1_Up",
                       iSL_Sen_Val1_Down := "S1_R1_Sen_Val1_Down",
                       iSL_Sen_Val2_Up := "S1_R1_Sen_Val2_Up",
                       iSL_Sen_Val2_Down := "S1_R1_Sen_Val2_Down",
                       iSR_Sen_Val1_Up := "S1_R2_Sen_Val1_Up",
                       iSR_Sen_Val1_Down := "S1_R2_Sen_Val1_Down",
                       iSR_Sen_Val2_Up := "S1_R2_Sen_Val2_Up",
                       iSR_Sen_Val2_Down := "S1_R2_Sen_Val2_Down",
                       iSL_Distance := "iS1L_Distance_Value",
                       iSR_Correct := 8,
                       iSR_Distance := "iS1R_Distance_Value",
                       HWIdentSL := "S1R1M~Module_I_O_(05_words)_1",
                       HWIdentSR := "S1R2M~Module_I_O_(05_words)_1",
                       Reset_Drive := "HMI_SideShifter_1".Reset_Drives OR "S5_Button_ST01_ST02",
                       Reset_Hydro := "HMI_SideShifter_1".Reset_Hydro,
                       iSL_Drive_Param := "Side_MOVIKIT".S1_R1_PI,
                       iSR_Drive_Param := "Side_MOVIKIT".S1_R2_PI,
                       oSL_Drive_Param := "Side_MOVIKIT".S1_R1_PO,
                       oSR_Drive_Param := "Side_MOVIKIT".S1_R2_PO,
                       oSL_Valve_Up => "S1_R1_Valve_Up",
                       oSL_Valve_Down => "S1_R1_Valve_Down",
                       oSL_Hydraulic_Unit => "S1_R1_Hydraulic_Unit",
                       oSR_Valve_Up => "S1_R2_Valve_Up",
                       oSR_Valve_Down => "S1_R2_Valve_Down",
                       oSR_Hydraulic_Unit => "S1_R2_Hydraulic_Unit",
                       oHydraulic_Status_LED_UP_1 => "Sz7_Button_LED_SS_Up",
                       oHydraulic_Status_LED_UP_2 => "S5_Button_LED_SS1_Up",
                       oHydraulic_Status_LED_DOWN_1 => "Sz7_Button_LED_SS_Down",
                       oHydraulic_Status_LED_DOWN_2 => "S5_Button_LED_SS1_Down",
                       oST1_1_Move_Flag => "S5_Button_LED_ST35",
                       oST1_2_Move_Flag => "Sz7_Button_LED_SS_Drive_ST35",
                       oST2_1_Move_Flag => "S5_Button_LED_ST02",
                       oST2_2_Move_Flag => "Sz7_Button_LED_SS_Drive_ST02",
                       oST3_1_Move_flag => "S5_Button_LED_ST03",
                       oST3_2_Move_Flag => "Sz7_Button_LED_SS_Drive_ST03",
                       oST4_1_Move_Flag => "S5_Button_LED_ST04",
                       oST4_2_Move_Flag => "Sz7_Button_LED_SS_Drive_ST04");
END_REGION

REGION Network 3: Pallet Circulation
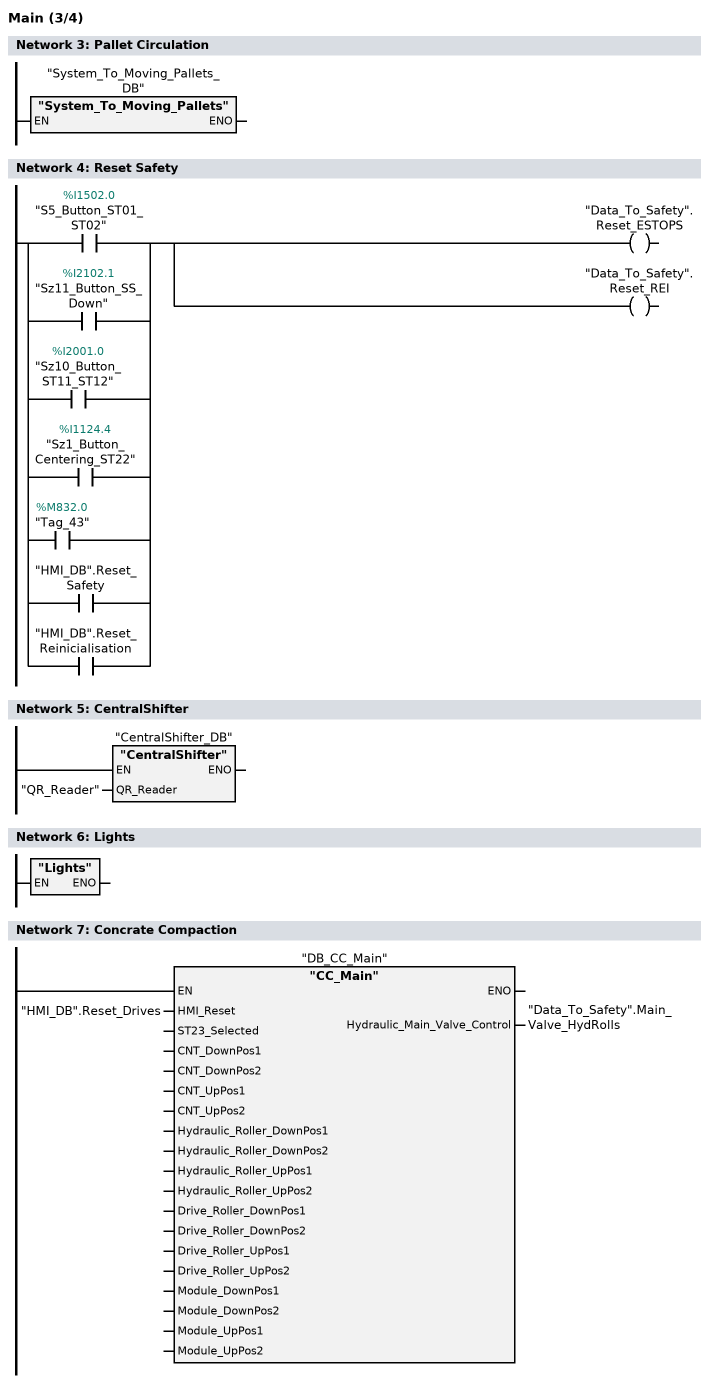
   RUNG wire#powerrail
      "System_To_Moving_Pallets_DB"()
   END_RUNG
   // the same network as SCL:
   "System_To_Moving_Pallets_DB"();   // "System_To_Moving_Pallets"
END_REGION

REGION Network 4: Reset Safety
   RUNG wire#powerrail
      Contact( "S5_Button_ST01_ST02" )
      wire#w1
      Coil( "Data_To_Safety".Reset_ESTOPS )
   END_RUNG
   RUNG wire#powerrail
      Contact( "Sz11_Button_SS_Down" )
   END_RUNG wire#w1
   RUNG wire#powerrail
      Contact( "Sz10_Button_ST11_ST12" )
   END_RUNG wire#w1
   RUNG wire#powerrail
      Contact( "Sz1_Button_Centering_ST22" )
   END_RUNG wire#w1
   RUNG wire#powerrail
      Contact( "Tag_43" )
   END_RUNG wire#w1
   RUNG wire#powerrail
      Contact( "HMI_DB".Reset_Safety )
   END_RUNG wire#w1
   RUNG wire#powerrail
      Contact( "HMI_DB".Reset_Reinicialisation )
   END_RUNG wire#w1
   RUNG wire#w1
      Coil( "Data_To_Safety".Reset_REI )
   END_RUNG
   // the same network as SCL:
   "Data_To_Safety".Reset_ESTOPS := "S5_Button_ST01_ST02" OR "Sz11_Button_SS_Down" OR "Sz10_Button_ST11_ST12" OR "Sz1_Button_Centering_ST22" OR "Tag_43" OR "HMI_DB".Reset_Safety OR "HMI_DB".Reset_Reinicialisation;
   "Data_To_Safety".Reset_REI := "Data_To_Safety".Reset_ESTOPS;
END_REGION

REGION Network 5: CentralShifter
   RUNG wire#powerrail
      "CentralShifter_DB"(QR_Reader := "QR_Reader")
   END_RUNG
   // the same network as SCL:
   "CentralShifter_DB"(QR_Reader := "QR_Reader");   // "CentralShifter"
END_REGION

REGION Network 6: Lights
   RUNG wire#powerrail
      "Lights"()
   END_RUNG
   // the same network as SCL:
   "Lights"();
END_REGION

REGION Network 7: Concrate Compaction
   RUNG wire#powerrail
      "DB_CC_Main"(HMI_Reset := "HMI_DB".Reset_Drives, ST23_Selected :=, CNT_DownPos1 :=, CNT_DownPos2 :=, CNT_UpPos1 :=, CNT_UpPos2 :=, Hydraulic_Roller_DownPos1 :=, Hydraulic_Roller_DownPos2 :=, Hydraulic_Roller_UpPos1 :=, Hydraulic_Roller_UpPos2 :=, Drive_Roller_DownPos1 :=, Drive_Roller_DownPos2 :=, Drive_Roller_UpPos1 :=, Drive_Roller_UpPos2 :=, Module_DownPos1 :=, Module_DownPos2 :=, Module_UpPos1 :=, Module_UpPos2 :=, Hydraulic_Main_Valve_Control => "Data_To_Safety".Main_Valve_HydRolls)
   END_RUNG
   // the same network as SCL:
   "DB_CC_Main"(HMI_Reset := "HMI_DB".Reset_Drives,   // "CC_Main"
                Hydraulic_Main_Valve_Control => "Data_To_Safety".Main_Valve_HydRolls);
END_REGION

REGION Network 8: Oil
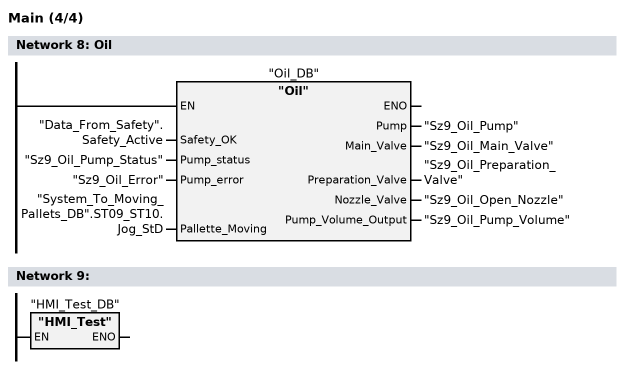
   RUNG wire#powerrail
      "Oil_DB"(Safety_OK := "Data_From_Safety".Safety_Active, Pump_status := "Sz9_Oil_Pump_Status", Pump_error := "Sz9_Oil_Error", Pallette_Moving := "System_To_Moving_Pallets_DB".ST09_ST10.Jog_StD, Pump => "Sz9_Oil_Pump", Main_Valve => "Sz9_Oil_Main_Valve", Preparation_Valve => "Sz9_Oil_Preparation_Valve", Nozzle_Valve => "Sz9_Oil_Open_Nozzle", Pump_Volume_Output => "Sz9_Oil_Pump_Volume")
   END_RUNG
   // the same network as SCL:
   "Oil_DB"(Safety_OK := "Data_From_Safety".Safety_Active,   // "Oil"
            Pump_status := "Sz9_Oil_Pump_Status",
            Pump_error := "Sz9_Oil_Error",
            Pallette_Moving := "System_To_Moving_Pallets_DB".ST09_ST10.Jog_StD,
            Pump => "Sz9_Oil_Pump",
            Main_Valve => "Sz9_Oil_Main_Valve",
            Preparation_Valve => "Sz9_Oil_Preparation_Valve",
            Nozzle_Valve => "Sz9_Oil_Open_Nozzle",
            Pump_Volume_Output => "Sz9_Oil_Pump_Volume");
END_REGION

REGION Network 9
   RUNG wire#powerrail
      "HMI_Test_DB"()
   END_RUNG
   // the same network as SCL:
   "HMI_Test_DB"();   // "HMI_Test"
END_REGION
END_ORGANIZATION_BLOCK

